          (** Set limits to all devices in the group **)
          IF GVL.UseTempGroupInputs AND (baseIdx - 10) + 6 < SIZEOF(GVL.TempGroupInput) / SIZEOF(GVL.TempGroupInput[0]) THEN
            THIS^.VoutSetMin[devIdx] := GVL.TempGroupInput[(baseIdx - 10) + 3];
            THIS^.VoutSetMax[devIdx] := GVL.TempGroupInput[(baseIdx - 10) + 4];
            THIS^.IoutSetMin[devIdx] := GVL.TempGroupInput[(baseIdx - 10) + 5];
            THIS^.IoutSetMax[devIdx] := MIN(GVL.TempGroupInput[(baseIdx - 10) + 6], GVL.GroupCapacity[groupIdx]);
          ELSE
            THIS^.VoutSetMin[devIdx] := GVL.NumericInput[baseIdx + 3]; (** GroupVoutSetMin **)
            THIS^.VoutSetMax[devIdx] := GVL.NumericInput[baseIdx + 4]; (** GroupVoutSetMax **)
            THIS^.IoutSetMin[devIdx] := GVL.NumericInput[baseIdx + 5]; (** GroupIoutSetMin **)
            THIS^.IoutSetMax[devIdx] := MIN(GVL.NumericInput[baseIdx + 6], GVL.GroupCapacity[groupIdx]); (** GroupIoutSetMax, constrained by min(GroupIoutSetMax, GroupCapacity) **)
          END_IF;
          
          (** Queue commands for group flags if changed **)
          IF GVL.Direction[devIdx] <> THIS^.LastDirection[devIdx] THEN
            IF THIS^.ApplyCommands(devIdx, GVL_Constant.CMD_DIRECTION_CTRL, BOOL_TO_UINT(GVL.Direction[devIdx])) THEN (** CMD_DIRECTION_CTRL **)
              THIS^.LastDirection[devIdx] := GVL.Direction[devIdx];
            END_IF;
          END_IF;
          
          IF GVL.OperationOn[devIdx] <> THIS^.LastOperationOn[devIdx] THEN
            IF THIS^.ApplyCommands(devIdx, GVL_Constant.CMD_OPERATION, BOOL_TO_UINT(GVL.OperationOn[devIdx])) THEN (** CMD_OPERATION **)
              THIS^.LastOperationOn[devIdx] := GVL.OperationOn[devIdx];
            END_IF;
          END_IF;
        END_IF;
      END_FOR;
    END_IF;
  END_IF;
END_FOR;

(** Process device inputs and queue control commands **)
FOR devIdx := 0 TO 19 DO
  baseIdx := 38 + (devIdx * 7); (** Device inputs start at 38 **)
  
  (** Read device setpoints and flags **)
  IF baseIdx + 6 < SIZEOF(GVL.NumericInput) / SIZEOF(GVL.NumericInput[0]) THEN
    (** Set setpoints for non-master devices or in maintenance mode **)
    IF GVL.UseTempBus1Direct AND devIdx <= 3 THEN
      GVL.VoutSetpoint[devIdx] := UINT_TO_REAL(GVL.TempBus1VoutSetpoint[devIdx]); (** Temp Bus1 VoutSetpoint **)
      GVL.IoutSetpoint[devIdx] := UINT_TO_REAL(GVL.TempBus1IoutSetpoint[devIdx]); (** Temp Bus1 IoutSetpoint **)
    ELSIF maintenanceMode OR devIdx < 4 OR GVL.GroupMembership[devIdx] = -1 OR NOT (GVL.GroupMaster[GVL.GroupMembership[devIdx]] = devIdx) THEN
      GVL.VoutSetpoint[devIdx] := UINT_TO_REAL(GVL.NumericInput[baseIdx]); (** VoutSetpoint **)
      GVL.IoutSetpoint[devIdx] := UINT_TO_REAL(GVL.NumericInput[baseIdx + 1]); (** IoutSetpoint **)
    END_IF;
    IF GVL.UseTempBus1Direct AND devIdx <= 3 THEN
      flags := GVL.TempBus1Flags[devIdx]; (** Temp Bus1 device flags **)
    ELSE
      flags := GVL.NumericInput[baseIdx + 2]; (** Device flags **)
    END_IF;
    
    (** Set device flags in maintenance mode or for devices 0-3 or non-master devices **)
    IF GVL.UseTempBus1Direct AND devIdx <= 3 THEN
      GVL.Voltage[devIdx] := (flags AND 16#0008) <> 0; (** Bit 3: DeviceMode Voltage **)
      GVL.Current[devIdx] := (flags AND 16#0004) <> 0; (** Bit 2: DeviceMode Current **)
      GVL.Standby[devIdx] := NOT (GVL.Voltage[devIdx] OR GVL.Current[devIdx]); (** Standby when neither Voltage nor Current **)
      GVL.Direction[devIdx] := (flags AND 16#0001) <> 0; (** Bit 0: Direction **)
      GVL.OperationOn[devIdx] := (flags AND 16#0002) <> 0; (** Bit 1: OperationOn **)
      GVL.OutputOn[devIdx] := (flags AND 16#0010) <> 0; (** Bit 4: OutputOn **)
    ELSIF maintenanceMode OR devIdx < 4 OR GVL.GroupMembership[devIdx] = -1 OR NOT (GVL.GroupMaster[GVL.GroupMembership[devIdx]] = devIdx) THEN
      GVL.Voltage[devIdx] := (flags AND 16#0008) <> 0; (** Bit 3: DeviceMode Voltage **)
      GVL.Current[devIdx] := (flags AND 16#0004) <> 0; (** Bit 2: DeviceMode Current **)
      GVL.Standby[devIdx] := NOT (GVL.Voltage[devIdx] OR GVL.Current[devIdx]); (** Standby when neither Voltage nor Current **)
      GVL.Direction[devIdx] := (flags AND 16#0001) <> 0; (** Bit 0: Direction **)
      GVL.OperationOn[devIdx] := (flags AND 16#0002) <> 0; (** Bit 1: OperationOn **)
      GVL.OutputOn[devIdx] := (flags AND 16#0010) <> 0; (** Bit 4: OutputOn **)
    END_IF;
    GVL.OrangeStop[devIdx] := (flags AND 16#0020) <> 0; (** Bit 5: OrangeStop **)
    GVL.RedStop[devIdx] := (flags AND 16#0040) <> 0; (** Bit 6: RedStop **)
    GVL.EStop[devIdx] := (flags AND 16#0080) <> 0; (** Bit 7: EStop **)
  END_IF;

  (** Queue direction command if requested direction differs from device feedback **)
  IF (GVL.UseTempBus1Direct AND devIdx <= 3 AND GVL.Direction[devIdx] <> THIS^.LastDirection[devIdx]) OR
     (NOT (GVL.UseTempBus1Direct AND devIdx <= 3) AND (GVL.Direction[devIdx] <> ((GVL.DeviceSystemFlags[devIdx] AND 16#0008) <> 0) OR 
     GVL.Direction[devIdx] <> THIS^.LastDirection[devIdx])) THEN
    IF THIS^.ApplyCommands(devIdx, GVL_Constant.CMD_DIRECTION_CTRL, BOOL_TO_UINT(GVL.Direction[devIdx])) THEN (** CMD_DIRECTION_CTRL **)
      THIS^.LastDirection[devIdx] := GVL.Direction[devIdx];
    END_IF;
  END_IF;

  (** Queue operation command **)
  IF GVL.OperationOn[devIdx] <> THIS^.LastOperationOn[devIdx] THEN
    IF THIS^.ApplyCommands(devIdx, GVL_Constant.CMD_OPERATION, BOOL_TO_UINT(GVL.OperationOn[devIdx])) THEN (** CMD_OPERATION **)
      THIS^.LastOperationOn[devIdx] := GVL.OperationOn[devIdx];
    END_IF;
  END_IF;

  (** Queue setpoint commands based on DeviceMode and Direction **)
  IF GVL.Standby[devIdx] THEN
    (** Standby mode **)
    IF THIS^.LastVoutSetpoint[devIdx] <> 0 THEN
      IF GVL.Direction[devIdx] THEN
        IF THIS^.ApplyCommands(devIdx, GVL_Constant.CMD_REVERSE_VOUT_SET, 0) THEN (** CMD_REVERSE_VOUT_SET, 0 **)
          GVL.VoutSetRev[devIdx] := 0.0; (** Clear reverse Vout setpoint **)
          THIS^.LastVoutSetpoint[devIdx] := 0;
        END_IF;
      ELSE
        IF THIS^.ApplyCommands(devIdx, GVL_Constant.CMD_VOUT_SET, 0) THEN (** CMD_VOUT_SET, 0 **)
          GVL.VoutSetpoint[devIdx] := 0.0; (** Clear forward Vout setpoint **)
          THIS^.LastVoutSetpoint[devIdx] := 0;
        END_IF;
      END_IF;
    END_IF;
    IF THIS^.LastIoutSetpoint[devIdx] <> 0 THEN
      IF GVL.Direction[devIdx] THEN
        IF THIS^.ApplyCommands(devIdx, GVL_Constant.CMD_REVERSE_IOUT_SET, 0) THEN (** CMD_REVERSE_IOUT_SET, 0 **)
          GVL.IoutSetRev[devIdx] := 0.0; (** Clear reverse Iout setpoint **)
          THIS^.LastIoutSetpoint[devIdx] := 0;
        END_IF;
      ELSE
        IF THIS^.ApplyCommands(devIdx, GVL_Constant.CMD_IOUT_SET, 0) THEN (** CMD_IOUT_SET, 0 **)
          GVL.IoutSetpoint[devIdx] := 0.0; (** Clear forward Iout setpoint **)
          THIS^.LastIoutSetpoint[devIdx] := 0;
        END_IF;
      END_IF;
    END_IF;
  ELSIF GVL.Current[devIdx] THEN
    (** Current mode **)
    setpointIout := MIN(MAX(GVL.IoutSetpoint[devIdx]/100, UINT_TO_REAL(THIS^.IoutSetMin[devIdx])), UINT_TO_REAL(THIS^.IoutSetMax[devIdx])); (** Clamp in native units **)
    IF devIdx <= 3 THEN
      clampedIout := REAL_TO_UINT(setpointIout * 10.0);   (** DPU F=0.1 **)
    ELSE
      factorNibble := SHR((GVL.VoutScale[devIdx] AND 16#00F0), 4);
      CASE factorNibble OF
        16#4: clampedIout := REAL_TO_UINT(setpointIout * 1000.0);
        16#5: clampedIout := REAL_TO_UINT(setpointIout * 100.0);
        16#6: clampedIout := REAL_TO_UINT(setpointIout * 10.0);
        16#7: clampedIout := REAL_TO_UINT(setpointIout);
        16#8: clampedIout := REAL_TO_UINT(setpointIout * 0.1);
        16#9: clampedIout := REAL_TO_UINT(setpointIout * 0.01);
        ELSE clampedIout := REAL_TO_UINT(setpointIout * 100.0);
      END_CASE;
    END_IF;
    IF clampedIout <> THIS^.LastIoutSetpoint[devIdx] THEN
      IF GVL.Direction[devIdx] THEN
        IF THIS^.ApplyCommands(devIdx, GVL_Constant.CMD_REVERSE_IOUT_SET, clampedIout) THEN (** CMD_REVERSE_IOUT_SET **)
          THIS^.LastIoutSetpoint[devIdx] := clampedIout;
        END_IF;
      ELSE
        IF THIS^.ApplyCommands(devIdx, GVL_Constant.CMD_IOUT_SET, clampedIout) THEN (** CMD_IOUT_SET **)
          THIS^.LastIoutSetpoint[devIdx] := clampedIout;
        END_IF;
      END_IF;
    END_IF;
  ELSIF GVL.Voltage[devIdx] THEN
    (** Voltage mode **)
    setpointVout := MIN(MAX(GVL.VoutSetpoint[devIdx]/100, UINT_TO_REAL(THIS^.VoutSetMin[devIdx])), UINT_TO_REAL(THIS^.VoutSetMax[devIdx])); (** Clamp in native units **)
    IF devIdx <= 3 THEN
      clampedVout := REAL_TO_UINT(setpointVout * 10.0);   (** DPU F=0.1 **)
    ELSE
      factorNibble := GVL.VoutScale[devIdx] AND 16#000F;
      CASE factorNibble OF
        16#4: clampedVout := REAL_TO_UINT(setpointVout * 1000.0);
        16#5: clampedVout := REAL_TO_UINT(setpointVout * 100.0);
        16#6: clampedVout := REAL_TO_UINT(setpointVout * 10.0);
        16#7: clampedVout := REAL_TO_UINT(setpointVout);
        16#8: clampedVout := REAL_TO_UINT(setpointVout * 0.1);
        16#9: clampedVout := REAL_TO_UINT(setpointVout * 0.01);
        ELSE clampedVout := REAL_TO_UINT(setpointVout * 100.0);
      END_CASE;
    END_IF;
    IF clampedVout <> THIS^.LastVoutSetpoint[devIdx] THEN
      IF GVL.Direction[devIdx] THEN
        IF THIS^.ApplyCommands(devIdx, GVL_Constant.CMD_REVERSE_VOUT_SET, clampedVout) THEN (** CMD_REVERSE_VOUT_SET **)
          THIS^.LastVoutSetpoint[devIdx] := clampedVout;
        END_IF;
      ELSE
        IF THIS^.ApplyCommands(devIdx, GVL_Constant.CMD_VOUT_SET, clampedVout) THEN (** CMD_VOUT_SET **)
          THIS^.LastVoutSetpoint[devIdx] := clampedVout;
        END_IF;
      END_IF;
    END_IF;
  END_IF;
END_FOR;
END_METHOD

METHOD ReadLimits
VAR
  devIdx : INT;                            (* Device index *)
  baseIdx : INT;                           (* Base index for device inputs *)
  inputIdx : INT;                          (* Base index for group inputs *)
  groupIdx : INT;                          (* Group index *)
  masterIdx : INT;                         (* Master device index *)
  maintenanceMode : BOOL;                  (* Maintenance mode status *)
  tempBase : INT;                          (* Temp: offset into TempGroupInput array *)
END_VAR

(* Comment Section: GVL.NumericInput Mapping for ReadLimits *)
(* This method reads individual setpoints/limits for all devices and applies *)
(* group-level setpoints/limits to the master device in normal mode. Group limits *)
(* (e.g., GroupIoutSetMax) are constrained by GVL.GroupCapacity, set by GroupManager *)
(* based on healthy units. GVL.GroupMaster serves as the group device index, *)
(* enabling groups when valid (4-19). *)

(* GVL.NumericInput Mapping *)
(* 0-4: System-Level Inputs *)
(*   0: GVL.SystemAlarms *)
(*   1: System Flags (maintenanceMode read here) *)
(*   2: Morphee Signal *)
(*   3-4: Reserved *)
(* 5-9: Unallocated *)
(* 10-37: Group Inputs (4 groups x 7 inputs) *)
(*   - For groupIdx = 0 TO 3, baseIdx = 10 + (groupIdx * 7): *)
(*     baseIdx: GroupVoutSetpoint *)
(*     baseIdx + 1: GroupIoutSetpoint *)
(*     baseIdx + 2: Group Flags *)
(*     baseIdx + 3: GroupVoutSetMin *)
(*     baseIdx + 4: GroupVoutSetMax *)
(*     baseIdx + 5: GroupIoutSetMin *)
(*     baseIdx + 6: GroupIoutSetMax *)
(*   - Applied to master device here if valid *)
(* 38-177: Device Inputs (20 devices x 7 inputs) *)
(*   - For devIdx = 0 TO 19, baseIdx = 38 + (devIdx * 7): *)
(*     baseIdx: VoutSetpoint *)
(*     baseIdx + 1: IoutSetpoint *)
(*     baseIdx + 2: Flags *)
(*     baseIdx + 3: VoutSetMin *)
(*     baseIdx + 4: VoutSetMax *)
(*     baseIdx + 5: IoutSetMin *)
(*     baseIdx + 6: IoutSetMax *)
(* 178+: Unallocated *)

(* Read maintenance mode *)
maintenanceMode := (GVL.NumericInput[1] AND 16#0001) <> 0; (* Index 1, bit 0 *)

(* Set individual device setpoints and limits *)
FOR devIdx := 0 TO 19 DO
  baseIdx := 38 + (devIdx * 7);
  IF baseIdx + 6 < SIZEOF(GVL.NumericInput) / SIZEOF(GVL.NumericInput[0]) THEN
    IF GVL.UseTempBus1Direct AND devIdx <= 3 THEN
      VoutSetpoint[devIdx] := GVL.TempBus1VoutSetpoint[devIdx];
      IoutSetpoint[devIdx] := GVL.TempBus1IoutSetpoint[devIdx];
      VoutSetMin[devIdx] := GVL.TempBus1VoutSetMin[devIdx] / 100;
      VoutSetMax[devIdx] := GVL.TempBus1VoutSetMax[devIdx] / 100;
      IoutSetMin[devIdx] := GVL.TempBus1IoutSetMin[devIdx] / 100;
      IoutSetMax[devIdx] := GVL.TempBus1IoutSetMax[devIdx] / 100;
    ELSE
      VoutSetpoint[devIdx] := GVL.NumericInput[baseIdx];
      IoutSetpoint[devIdx] := GVL.NumericInput[baseIdx + 1];
      VoutSetMin[devIdx] := GVL.NumericInput[baseIdx + 3];
      VoutSetMax[devIdx] := GVL.NumericInput[baseIdx + 4];
      IoutSetMin[devIdx] := GVL.NumericInput[baseIdx + 5];
      IoutSetMax[devIdx] := GVL.NumericInput[baseIdx + 6];
    END_IF;
  END_IF;

  (* Apply group-level setpoints and limits to master in normal mode *)
  IF NOT maintenanceMode AND devIdx >= 4 THEN
    FOR groupIdx := 0 TO 3 DO
      masterIdx := GVL.GroupMaster[groupIdx];
      IF masterIdx >= 4 AND masterIdx <= 19 AND NOT GVL.SafetyShutdown[masterIdx] THEN
        CASE groupIdx OF
          0: inputIdx := 10; (* LVLA1 *)
          1: inputIdx := 17; (* LVLA2 *)
          2: inputIdx := 24; (* LVLA3 *)
          3: inputIdx := 31; (* LVLA4 *)
        END_CASE;
        IF devIdx = masterIdx THEN
          IF inputIdx + 6 < SIZEOF(GVL.NumericInput) / SIZEOF(GVL.NumericInput[0]) THEN
            IF GVL.UseTempGroupInputs THEN
              tempBase := inputIdx - 10; (* Map group base (10..) to TempGroupInput (0..) *)
              IF tempBase >= 0 AND tempBase + 6 < SIZEOF(GVL.TempGroupInput) / SIZEOF(GVL.TempGroupInput[0]) THEN
                VoutSetpoint[masterIdx] := GVL.TempGroupInput[tempBase];
                IoutSetpoint[masterIdx] := GVL.TempGroupInput[tempBase + 1];
                VoutSetMin[masterIdx] := GVL.TempGroupInput[tempBase + 3];
                VoutSetMax[masterIdx] := GVL.TempGroupInput[tempBase + 4];
                IoutSetMin[masterIdx] := GVL.TempGroupInput[tempBase + 5];
                IoutSetMax[masterIdx] := MIN(GVL.TempGroupInput[tempBase + 6], GVL.GroupCapacity[groupIdx]); (* Constrain by capacity *)
              END_IF;
            ELSE
              VoutSetpoint[masterIdx] := GVL.NumericInput[inputIdx];
              IoutSetpoint[masterIdx] := GVL.NumericInput[inputIdx + 1];
              VoutSetMin[masterIdx] := GVL.NumericInput[inputIdx + 3];
              VoutSetMax[masterIdx] := GVL.NumericInput[inputIdx + 4];
              IoutSetMin[masterIdx] := GVL.NumericInput[inputIdx + 5];
              IoutSetMax[masterIdx] := MIN(GVL.NumericInput[inputIdx + 6], GVL.GroupCapacity[groupIdx]); (* Constrain by capacity *)
            END_IF;
          END_IF;
        END_IF;
      END_IF;
    END_FOR;
  END_IF;
END_FOR;
END_METHOD

METHOD UpdateOutputs
VAR
  devIdx : INT;                            (* Device index *)
  baseIdx : INT;                           (* Base index for output array *)
  systemAlarms : DWORD;                    (* System alarms for output *)
  maintenanceMode : BOOL;                  (* Maintenance mode status *)
  cmdId : BYTE;                            (* Command ID for init data *)
  cmdOffset : INT;                         (* Command offset for init frame *)
  i : INT;                                 (* Loop variable for commands *)
  j : INT;                                 (* Loop variable for data pairs *)
  idx : INT;                               (* Output array index *)
  watchDog : BOOL;                         (* Watchdog toggle for output *)
  updatingInMorpheeTableInprogress : Bool := FALSE;
  groupIdx : INT;                          (* Group index *)
  masterIdx : INT;                         (* Master device index *)
  groupBase : INT;                         (* Base index for group devices *)
  opCount : UINT;                          (* Count of devices with OperationOn *)
  outCount : UINT;                         (* Count of devices with OutputOn *)
  initTimeoutCounter : UINT;               (* Counter for forced init exit *)
  commandCount : UINT;                     (* Commands per cycle *)
  commandArray : ARRAY[0..8] OF BYTE := [16#80, 16#81, 16#82, 16#83, 16#84, 16#85, 16#86, 16#87, 16#88];
  commandIndex : INT;
  upperBound : INT;                        (* Upper bound for FOR loop *)
	scaledVin: INT; (** Scaled input voltage **)
	scaledVout: UINT; (** Scaled output voltage **)
	scaledIout: UINT; (** Scaled current **)
	scaledTemp: UINT; (** Scaled temperature **)
	scaledFanSpeed1: INT; (** Scaled fan speed 1 **)
	scaledFanSpeed2: INT; (** Scaled fan speed 2 **)
	scaledIin: INT; (** Scaled input current **)
	tempScale: UINT; (** Temporary variable for scaling factor extraction **)
	scaleValue: UINT; (** Extracted 4-bit scaling value **)
 
END_VAR
(* One-time reset of GVL variables *)
IF GVL.FirstRun THEN
    FOR devIdx := 0 TO 19 DO
        GVL.Voltage[devIdx] := FALSE;
        GVL.Current[devIdx] := FALSE;
        GVL.Standby[devIdx] := FALSE;
        GVL.OperationOn[devIdx] := FALSE;
        GVL.Direction[devIdx] := FALSE;
        GVL.OutputOn[devIdx] := FALSE;
        GVL.OrangeStop[devIdx] := FALSE;
        GVL.RedStop[devIdx] := FALSE;
        GVL.EStop[devIdx] := FALSE;
        GVL.Vin[devIdx] := 0;
        GVL.Vout[devIdx] := 0;
        GVL.Iout[devIdx] := 0;
        GVL.Temperature[devIdx] := 0;
        GVL.FanSpeed1[devIdx] := 0;
        GVL.FanSpeed2[devIdx] := 0;
        GVL.Iin[devIdx] := 0;
        GVL.FaultStatus[devIdx] := 0;
        GVL.TemperatureFaultHigh[devIdx] := FALSE;
        CanCtrlConfigured[devIdx] := FALSE;
    END_FOR;
    GVL.FirstRun := FALSE;
END_IF;

watchDog := NOT watchDog;


// Detect Morphee initialization request (GVL.NumericInput[2] changes)
IF GVL.NumericInput[2] <> LastMorpheeSignal AND NOT updatingInMorpheeTableInprogress THEN
    LastMorpheeSignal := DWORD_TO_UINT(GVL.NumericInput[2]);
    CASE GVL.NumericInput[2] OF
        1..6: // Morphee requests initialization cycles 1 to 6
            IsInitPhase := TRUE;
            InitCycle := DWORD_TO_UINT(GVL.NumericInput[2]);
            initTimeoutCounter := 0;
            InitTimeout(IN := FALSE);
        100: // Morphee signals completion
            IsInitPhase := FALSE;
            InitCycle := 0;
            initTimeoutCounter := 0;
            InitTimeout(IN := FALSE);
    END_CASE;
END_IF;

(* In temporary setpoint test mode, keep normal output update path active. *)
IF GVL.UseTempGroupInputs THEN
  IsInitPhase := FALSE;
  InitCycle := 0;
END_IF;

// Initialization phase logic
IF IsInitPhase THEN
    initTimeoutCounter := initTimeoutCounter + 1;
    // Remove strict timeout to ensure all cycles complete
    // IF initTimeoutCounter > 1000 THEN
    //     IsInitPhase := FALSE;
    //     InitCycle := 0;
    //     initTimeoutCounter := 0;
    //     InitTimeout(IN := FALSE);
    // END_IF;

    InitTimeout(IN := TRUE, PT := T#100MS);

    IF InitCycle > 0 AND IsInitPhase THEN
        updatingInMorpheeTableInprogress := TRUE;
        FOR devIdx := 0 TO 19 DO
            idx := devIdx * 6; // Base index for the device
            IF idx + 5 < 120 THEN // Ensure within array bounds
                CASE InitCycle OF
                    1: // 0x80 and 0x81 (bytes 0-11)
                        cmdId := 16#80;
                        baseIdx := 0;
                        IF baseIdx + 1 < 54 THEN
                            GVL.NumericOutput[idx] := SHL(TO_DWORD(cmdId), 24) OR SHL(TO_DWORD(devIdx), 16) OR SHL(TO_DWORD(GVL.MfrSerialPersistent[devIdx][baseIdx]), 8) OR TO_DWORD(GVL.MfrSerialPersistent[devIdx][baseIdx + 1]);
                            GVL.NumericOutput[idx + 1] := SHL(TO_DWORD(cmdId), 24) OR SHL(TO_DWORD(devIdx), 16) OR SHL(TO_DWORD(GVL.MfrSerialPersistent[devIdx][baseIdx + 2]), 8) OR TO_DWORD(GVL.MfrSerialPersistent[devIdx][baseIdx + 3]);
                            GVL.NumericOutput[idx + 2] := SHL(TO_DWORD(cmdId), 24) OR SHL(TO_DWORD(devIdx), 16) OR SHL(TO_DWORD(GVL.MfrSerialPersistent[devIdx][baseIdx + 4]), 8) OR TO_DWORD(GVL.MfrSerialPersistent[devIdx][baseIdx + 5]);
                        END_IF;
                        cmdId := 16#81;
                        baseIdx := 6;
                        IF baseIdx + 1 < 54 THEN
                            GVL.NumericOutput[idx + 3] := SHL(TO_DWORD(cmdId), 24) OR SHL(TO_DWORD(devIdx), 16) OR SHL(TO_DWORD(GVL.MfrSerialPersistent[devIdx][baseIdx]), 8) OR TO_DWORD(GVL.MfrSerialPersistent[devIdx][baseIdx + 1]);
                            GVL.NumericOutput[idx + 4] := SHL(TO_DWORD(cmdId), 24) OR SHL(TO_DWORD(devIdx), 16) OR SHL(TO_DWORD(GVL.MfrSerialPersistent[devIdx][baseIdx + 2]), 8) OR TO_DWORD(GVL.MfrSerialPersistent[devIdx][baseIdx + 3]);
                            GVL.NumericOutput[idx + 5] := SHL(TO_DWORD(cmdId), 24) OR SHL(TO_DWORD(devIdx), 16) OR SHL(TO_DWORD(GVL.MfrSerialPersistent[devIdx][baseIdx + 4]), 8) OR TO_DWORD(GVL.MfrSerialPersistent[devIdx][baseIdx + 5]);
                        END_IF;
                    2: // 0x82 and 0x83 (bytes 12-23)
                        cmdId := 16#82;
                        baseIdx := 12;
                        IF baseIdx + 1 < 54 THEN
                            GVL.NumericOutput[idx] := SHL(TO_DWORD(cmdId), 24) OR SHL(TO_DWORD(devIdx), 16) OR SHL(TO_DWORD(GVL.MfrSerialPersistent[devIdx][baseIdx]), 8) OR TO_DWORD(GVL.MfrSerialPersistent[devIdx][baseIdx + 1]);
                            GVL.NumericOutput[idx + 1] := SHL(TO_DWORD(cmdId), 24) OR SHL(TO_DWORD(devIdx), 16) OR SHL(TO_DWORD(GVL.MfrSerialPersistent[devIdx][baseIdx + 2]), 8) OR TO_DWORD(GVL.MfrSerialPersistent[devIdx][baseIdx + 3]);
                            GVL.NumericOutput[idx + 2] := SHL(TO_DWORD(cmdId), 24) OR SHL(TO_DWORD(devIdx), 16) OR SHL(TO_DWORD(GVL.MfrSerialPersistent[devIdx][baseIdx + 4]), 8) OR TO_DWORD(GVL.MfrSerialPersistent[devIdx][baseIdx + 5]);
                        END_IF;
                        cmdId := 16#83;
                        baseIdx := 18;
                        IF baseIdx + 1 < 54 THEN
                            GVL.NumericOutput[idx + 3] := SHL(TO_DWORD(cmdId), 24) OR SHL(TO_DWORD(devIdx), 16) OR SHL(TO_DWORD(GVL.MfrSerialPersistent[devIdx][baseIdx]), 8) OR TO_DWORD(GVL.MfrSerialPersistent[devIdx][baseIdx + 1]);
                            GVL.NumericOutput[idx + 4] := SHL(TO_DWORD(cmdId), 24) OR SHL(TO_DWORD(devIdx), 16) OR SHL(TO_DWORD(GVL.MfrSerialPersistent[devIdx][baseIdx + 2]), 8) OR TO_DWORD(GVL.MfrSerialPersistent[devIdx][baseIdx + 3]);
                            GVL.NumericOutput[idx + 5] := SHL(TO_DWORD(cmdId), 24) OR SHL(TO_DWORD(devIdx), 16) OR SHL(TO_DWORD(GVL.MfrSerialPersistent[devIdx][baseIdx + 4]), 8) OR TO_DWORD(GVL.MfrSerialPersistent[devIdx][baseIdx + 5]);
                        END_IF;
                    3: // 0x84 (bytes 24-29)
                        cmdId := 16#84;
                        baseIdx := 24;
                        IF baseIdx + 1 < 54 THEN
                            GVL.NumericOutput[idx] := SHL(TO_DWORD(cmdId), 24) OR SHL(TO_DWORD(devIdx), 16) OR SHL(TO_DWORD(GVL.MfrSerialPersistent[devIdx][baseIdx]), 8) OR TO_DWORD(GVL.MfrSerialPersistent[devIdx][baseIdx + 1]);
                            GVL.NumericOutput[idx + 1] := SHL(TO_DWORD(cmdId), 24) OR SHL(TO_DWORD(devIdx), 16) OR SHL(TO_DWORD(GVL.MfrSerialPersistent[devIdx][baseIdx + 2]), 8) OR TO_DWORD(GVL.MfrSerialPersistent[devIdx][baseIdx + 3]);
                            GVL.NumericOutput[idx + 2] := SHL(TO_DWORD(cmdId), 24) OR SHL(TO_DWORD(devIdx), 16) OR SHL(TO_DWORD(GVL.MfrSerialPersistent[devIdx][baseIdx + 4]), 8) OR TO_DWORD(GVL.MfrSerialPersistent[devIdx][baseIdx + 5]);
                        END_IF;
                    4: // 0x85 (bytes 30-35)
                        cmdId := 16#85;
                        baseIdx := 30;
                        IF baseIdx + 1 < 54 THEN
                            GVL.NumericOutput[idx] := SHL(TO_DWORD(cmdId), 24) OR SHL(TO_DWORD(devIdx), 16) OR SHL(TO_DWORD(GVL.MfrSerialPersistent[devIdx][baseIdx]), 8) OR TO_DWORD(GVL.MfrSerialPersistent[devIdx][baseIdx + 1]);
                            GVL.NumericOutput[idx + 1] := SHL(TO_DWORD(cmdId), 24) OR SHL(TO_DWORD(devIdx), 16) OR SHL(TO_DWORD(GVL.MfrSerialPersistent[devIdx][baseIdx + 2]), 8) OR TO_DWORD(GVL.MfrSerialPersistent[devIdx][baseIdx + 3]);
                            GVL.NumericOutput[idx + 2] := SHL(TO_DWORD(cmdId), 24) OR SHL(TO_DWORD(devIdx), 16) OR SHL(TO_DWORD(GVL.MfrSerialPersistent[devIdx][baseIdx + 4]), 8) OR TO_DWORD(GVL.MfrSerialPersistent[devIdx][baseIdx + 5]);
                        END_IF;
                    5: // 0x86 (bytes 36-41)
                        cmdId := 16#86;
                        baseIdx := 36;
                        IF baseIdx + 1 < 54 THEN
                            GVL.NumericOutput[idx] := SHL(TO_DWORD(cmdId), 24) OR SHL(TO_DWORD(devIdx), 16) OR SHL(TO_DWORD(GVL.MfrSerialPersistent[devIdx][baseIdx]), 8) OR TO_DWORD(GVL.MfrSerialPersistent[devIdx][baseIdx + 1]);
                            GVL.NumericOutput[idx + 1] := SHL(TO_DWORD(cmdId), 24) OR SHL(TO_DWORD(devIdx), 16) OR SHL(TO_DWORD(GVL.MfrSerialPersistent[devIdx][baseIdx + 2]), 8) OR TO_DWORD(GVL.MfrSerialPersistent[devIdx][baseIdx + 3]);
                            GVL.NumericOutput[idx + 2] := SHL(TO_DWORD(cmdId), 24) OR SHL(TO_DWORD(devIdx), 16) OR SHL(TO_DWORD(GVL.MfrSerialPersistent[devIdx][baseIdx + 4]), 8) OR TO_DWORD(GVL.MfrSerialPersistent[devIdx][baseIdx + 5]);
                        END_IF;
                    6: // 0x87 and 0x88 (bytes 42-53)
                        cmdId := 16#87;
                        baseIdx := 42;
                        IF baseIdx + 1 < 54 THEN
                            GVL.NumericOutput[idx] := SHL(TO_DWORD(cmdId), 24) OR SHL(TO_DWORD(devIdx), 16) OR SHL(TO_DWORD(GVL.MfrSerialPersistent[devIdx][baseIdx]), 8) OR TO_DWORD(GVL.MfrSerialPersistent[devIdx][baseIdx + 1]);
                            GVL.NumericOutput[idx + 1] := SHL(TO_DWORD(cmdId), 24) OR SHL(TO_DWORD(devIdx), 16) OR SHL(TO_DWORD(GVL.MfrSerialPersistent[devIdx][baseIdx + 2]), 8) OR TO_DWORD(GVL.MfrSerialPersistent[devIdx][baseIdx + 3]);
                            GVL.NumericOutput[idx + 2] := SHL(TO_DWORD(cmdId), 24) OR SHL(TO_DWORD(devIdx), 16) OR SHL(TO_DWORD(GVL.MfrSerialPersistent[devIdx][baseIdx + 4]), 8) OR TO_DWORD(GVL.MfrSerialPersistent[devIdx][baseIdx + 5]);
                        END_IF;
                        cmdId := 16#88;
                        baseIdx := 48;
                        IF baseIdx + 1 < 54 THEN
                            GVL.NumericOutput[idx + 3] := SHL(TO_DWORD(cmdId), 24) OR SHL(TO_DWORD(devIdx), 16) OR SHL(TO_DWORD(GVL.MfrSerialPersistent[devIdx][baseIdx]), 8) OR TO_DWORD(GVL.MfrSerialPersistent[devIdx][baseIdx + 1]);
                            GVL.NumericOutput[idx + 4] := SHL(TO_DWORD(cmdId), 24) OR SHL(TO_DWORD(devIdx), 16) OR SHL(TO_DWORD(GVL.MfrSerialPersistent[devIdx][baseIdx + 2]), 8) OR TO_DWORD(GVL.MfrSerialPersistent[devIdx][baseIdx + 3]);
                            GVL.NumericOutput[idx + 5] := SHL(TO_DWORD(cmdId), 24) OR SHL(TO_DWORD(devIdx), 16) OR SHL(TO_DWORD(GVL.MfrSerialPersistent[devIdx][baseIdx + 4]), 8) OR TO_DWORD(GVL.MfrSerialPersistent[devIdx][baseIdx + 5]);
                        END_IF;
                END_CASE;
            END_IF;
        END_FOR;
        updatingInMorpheeTableInprogress := FALSE;
    END_IF;
ELSE
    updatingInMorpheeTableInprogress := FALSE;
    InitTimeout(IN := FALSE);
    systemAlarms := UINT_TO_DWORD(GVL.SystemAlarms);
    maintenanceMode := (GVL.NumericInput[1] AND 16#0001) <> 0;

    FOR devIdx := 0 TO 19 DO
        baseIdx := devIdx * 5;
        // IF baseIdx < SIZEOF(GVL.NumericOutput) / SIZEOF(GVL.NumericOutput[0]) THEN
            (* Check for RedStop condition *)
            IF GVL.RedStop[devIdx] THEN
                GVL.Voltage[devIdx] := FALSE;
                GVL.Current[devIdx] := FALSE;
                GVL.Standby[devIdx] := TRUE;
                GVL.OperationOn[devIdx] := FALSE;
                GVL.Direction[devIdx] := FALSE;
                GVL.OutputOn[devIdx] := FALSE;
                GVL.OrangeStop[devIdx] := FALSE;
            END_IF;

            IF devIdx <= 3 THEN
              (* DPU fixed scaling from manual: VIN F=1, VOUT/IOUT/TEMP F=0.1, FAN F=1 *)
              scaledVin := GVL.Vin[devIdx];
              scaledVout := REAL_TO_UINT(UINT_TO_REAL(GVL.Vout[devIdx]) * 0.1);
            ELSE
              (* Scale GVL.Vin[devIdx] using VIN scaling factor, byte 1 bits 0-3 *)
              tempScale := GVL.VinScale[devIdx] AND 16#0F; (* Extract bits 0-3 *)
              IF tempScale = 16#4 THEN
                scaledVin := REAL_TO_UINT(UINT_TO_REAL(GVL.Vin[devIdx]) * 0.001);
              ELSIF tempScale = 16#5 THEN
                scaledVin := REAL_TO_UINT(UINT_TO_REAL(GVL.Vin[devIdx]) * 0.01);
              ELSIF tempScale = 16#6 THEN
                scaledVin := REAL_TO_UINT(UINT_TO_REAL(GVL.Vin[devIdx]) * 0.1);
              ELSIF tempScale = 16#7 THEN
                scaledVin := GVL.Vin[devIdx];
              ELSIF tempScale = 16#8 THEN
                scaledVin := REAL_TO_UINT(UINT_TO_REAL(GVL.Vin[devIdx]) * 10.0);
              ELSIF tempScale = 16#9 THEN
                scaledVin := REAL_TO_UINT(UINT_TO_REAL(GVL.Vin[devIdx]) * 100.0);
              ELSE
                scaledVin := REAL_TO_UINT(UINT_TO_REAL(GVL.Vin[devIdx]) * 0.1);
              END_IF;

              (* Scale GVL.Vout[devIdx] using VOUT scaling factor, byte 0 bits 0-3 *)
              tempScale := GVL.VoutScale[devIdx] AND 16#0F; (* Extract bits 0-3 *)
              IF tempScale = 16#4 THEN
                scaledVout := REAL_TO_UINT(UINT_TO_REAL(GVL.Vout[devIdx]) * 0.001);
              ELSIF tempScale = 16#5 THEN
                scaledVout := REAL_TO_UINT(UINT_TO_REAL(GVL.Vout[devIdx]) * 0.01);
              ELSIF tempScale = 16#6 THEN
                scaledVout := REAL_TO_UINT(UINT_TO_REAL(GVL.Vout[devIdx]) * 0.1);
              ELSIF tempScale = 16#7 THEN
                scaledVout := GVL.Vout[devIdx];
              ELSIF tempScale = 16#8 THEN
                scaledVout := REAL_TO_UINT(UINT_TO_REAL(GVL.Vout[devIdx]) * 10.0);
              ELSIF tempScale = 16#9 THEN
                scaledVout := REAL_TO_UINT(UINT_TO_REAL(GVL.Vout[devIdx]) * 100.0);
              ELSE
                scaledVout := REAL_TO_UINT(UINT_TO_REAL(GVL.Vout[devIdx]) * 0.1);
              END_IF;
            END_IF;

            IF GVL.Vin[devIdx] > 0 OR GVL.Vout[devIdx] > 0 THEN
              GVL.NumericOutput[baseIdx] := SHL(TO_DWORD(scaledVin), 16) OR TO_DWORD(scaledVout);
            ELSE
                GVL.NumericOutput[baseIdx] := 0;
            END_IF;

            IF devIdx <= 3 THEN
              scaledIout := REAL_TO_UINT(UINT_TO_REAL(GVL.Iout[devIdx]) * 0.1);
              scaledTemp := REAL_TO_UINT(UINT_TO_REAL(GVL.Temperature[devIdx]) * 0.1);
            ELSE
              (* Scale GVL.Iout[devIdx] using IOUT scaling factor, byte 0 bits 4-7 *)
              tempScale := GVL.VoutScale[devIdx] AND 16#F0; (* Mask bits 4-7 *)
              scaleValue := SHR(tempScale, 4); (* Shift right by 4 to get IOUT bits *)
              IF scaleValue = 16#4 THEN
                scaledIout := REAL_TO_UINT(UINT_TO_REAL(GVL.Iout[devIdx]) * 0.001);
              ELSIF scaleValue = 16#5 THEN
                scaledIout := REAL_TO_UINT(UINT_TO_REAL(GVL.Iout[devIdx]) * 0.01);
              ELSIF scaleValue = 16#6 THEN
                scaledIout := REAL_TO_UINT(UINT_TO_REAL(GVL.Iout[devIdx]) * 0.1);
              ELSIF scaleValue = 16#7 THEN
                scaledIout := GVL.Iout[devIdx];
              ELSIF scaleValue = 16#8 THEN
                scaledIout := REAL_TO_UINT(UINT_TO_REAL(GVL.Iout[devIdx]) * 10.0);
              ELSIF scaleValue = 16#9 THEN
                scaledIout := REAL_TO_UINT(UINT_TO_REAL(GVL.Iout[devIdx]) * 100.0);
              ELSE
                scaledIout := REAL_TO_UINT(UINT_TO_REAL(GVL.Iout[devIdx]) * 0.1);
              END_IF;

              (* Scale GVL.Temperature[devIdx] using TEMPERATURE_1 scaling factor, byte 2 bits 0-3 *)
              tempScale := GVL.TempScale[devIdx] AND 16#0F; (* Extract bits 0-3 *)
              IF tempScale = 16#4 THEN
                scaledTemp := REAL_TO_UINT(UINT_TO_REAL(GVL.Temperature[devIdx]) * 0.001);
              ELSIF tempScale = 16#5 THEN
                scaledTemp := REAL_TO_UINT(UINT_TO_REAL(GVL.Temperature[devIdx]) * 0.01);
              ELSIF tempScale = 16#6 THEN
                scaledTemp := REAL_TO_UINT(UINT_TO_REAL(GVL.Temperature[devIdx]) * 0.1);
              ELSIF tempScale = 16#7 THEN
                scaledTemp := GVL.Temperature[devIdx];
              ELSIF tempScale = 16#8 THEN
                scaledTemp := REAL_TO_UINT(UINT_TO_REAL(GVL.Temperature[devIdx]) * 10.0);
              ELSIF tempScale = 16#9 THEN
                scaledTemp := REAL_TO_UINT(UINT_TO_REAL(GVL.Temperature[devIdx]) * 100.0);
              ELSE
                scaledTemp := REAL_TO_UINT(UINT_TO_REAL(GVL.Temperature[devIdx]) * 0.1);
              END_IF;
            END_IF;

            (* Scale GVL.FanSpeed1[devIdx] and GVL.FanSpeed2[devIdx] using FAN_SPEED scaling factor, byte 1 bits 4-7 *)
            tempScale := GVL.VinScale[devIdx] AND 16#F0; (* Mask bits 4-7 *)
            scaleValue := SHR(tempScale, 4); (* Shift right by 4 to get FAN_SPEED bits *)
            IF scaleValue = 16#4 THEN
                scaledFanSpeed1 := REAL_TO_UINT(UINT_TO_REAL(GVL.FanSpeed1[devIdx]) * 0.001);
                scaledFanSpeed2 := REAL_TO_UINT(UINT_TO_REAL(GVL.FanSpeed2[devIdx]) * 0.001);
            ELSIF scaleValue = 16#5 THEN
                scaledFanSpeed1 := REAL_TO_UINT(UINT_TO_REAL(GVL.FanSpeed1[devIdx]) * 0.01);
                scaledFanSpeed2 := REAL_TO_UINT(UINT_TO_REAL(GVL.FanSpeed2[devIdx]) * 0.01);
            ELSIF scaleValue = 16#6 THEN
                scaledFanSpeed1 := REAL_TO_UINT(UINT_TO_REAL(GVL.FanSpeed1[devIdx]) * 0.1);
                scaledFanSpeed2 := REAL_TO_UINT(UINT_TO_REAL(GVL.FanSpeed2[devIdx]) * 0.1);
            ELSIF scaleValue = 16#7 THEN
                scaledFanSpeed1 := GVL.FanSpeed1[devIdx];
                scaledFanSpeed2 := GVL.FanSpeed2[devIdx];
            ELSIF scaleValue = 16#8 THEN
                scaledFanSpeed1 := REAL_TO_UINT(UINT_TO_REAL(GVL.FanSpeed1[devIdx]) * 10.0);
                scaledFanSpeed2 := REAL_TO_UINT(UINT_TO_REAL(GVL.FanSpeed2[devIdx]) * 10.0);
            ELSIF scaleValue = 16#9 THEN
                scaledFanSpeed1 := REAL_TO_UINT(UINT_TO_REAL(GVL.FanSpeed1[devIdx]) * 100.0);
                scaledFanSpeed2 := REAL_TO_UINT(UINT_TO_REAL(GVL.FanSpeed2[devIdx]) * 100.0);
            ELSE
                scaledFanSpeed1 := REAL_TO_UINT(UINT_TO_REAL(GVL.FanSpeed1[devIdx]) * 0.1);
                scaledFanSpeed2 := REAL_TO_UINT(UINT_TO_REAL(GVL.FanSpeed2[devIdx]) * 0.1);
            END_IF;

            (* Scale GVL.Iin[devIdx] using IIN scaling factor, byte 3 bits 0-3 *)
            tempScale := GVL.IinScale[devIdx] AND 16#0F; (* Extract bits 0-3 *)
            IF tempScale = 16#4 THEN
                scaledIin := REAL_TO_UINT(UINT_TO_REAL(GVL.Iin[devIdx]) * 0.001);
            ELSIF tempScale = 16#5 THEN
                scaledIin := REAL_TO_UINT(UINT_TO_REAL(GVL.Iin[devIdx]) * 0.01);
            ELSIF tempScale = 16#6 THEN
                scaledIin := REAL_TO_UINT(UINT_TO_REAL(GVL.Iin[devIdx]) * 0.1);
            ELSIF tempScale = 16#7 THEN
                scaledIin := GVL.Iin[devIdx];
            ELSIF tempScale = 16#8 THEN
                scaledIin := REAL_TO_UINT(UINT_TO_REAL(GVL.Iin[devIdx]) * 10.0);
            ELSIF tempScale = 16#9 THEN
                scaledIin := REAL_TO_UINT(UINT_TO_REAL(GVL.Iin[devIdx]) * 100.0);
            ELSE
                scaledIin := REAL_TO_UINT(UINT_TO_REAL(GVL.Iin[devIdx]) * 0.1);
            END_IF;

            GVL.NumericOutput[baseIdx + 1] := SHL(TO_DWORD(scaledIout), 16) OR TO_DWORD(scaledTemp);
            GVL.NumericOutput[baseIdx + 2] := SHL(TO_DWORD(scaledFanSpeed1), 16) OR TO_DWORD(scaledFanSpeed2);
            GVL.NumericOutput[baseIdx + 3] := SHL(TO_DWORD(GVL.FaultStatus[devIdx]), 16) OR 
                                              SHL(TO_DWORD(GVL.Direction[devIdx]), 0) OR 
                                              SHL(TO_DWORD(GVL.OperationOn[devIdx]), 1) OR 
                                              SHL(TO_DWORD(GVL.Current[devIdx]), 2) OR 
                                              SHL(TO_DWORD(GVL.Voltage[devIdx]), 3) OR 
                                              SHL(TO_DWORD(GVL.OutputOn[devIdx]), 4) OR 
                                              SHL(TO_DWORD(GVL.OrangeStop[devIdx]), 5) OR 
                                              SHL(TO_DWORD(GVL.RedStop[devIdx]), 6) OR 
                                              SHL(TO_DWORD(GVL.EStop[devIdx]), 7) OR 
                                              SHL(TO_DWORD(GVL.TemperatureFaultHigh[devIdx]), 8);
              GVL.NumericOutput[baseIdx + 4] := SHL(TO_DWORD(GVL.DeviceSystemFlags[devIdx]), 16);
        //END_IF;
    END_FOR;

    GVL.NumericOutput[100] := systemAlarms;
	 EL3174_Channel1_Alarm:=  EL3174_Channel1_value>(2.5*10)/32768;
 	 EL3174_Channel2_Alarm:=  EL3174_Channel2_value>(2.5*10)/32768;
 	 EL3174_Channel3_Alarm:=  EL3174_Channel3_value>(2.5*10)/32768;
	 EL3174_Channel4_Alarm:=  EL3174_Channel4_value>(2.5*10)/32768;
    GVL.NumericOutput[101] := SHL(TO_DWORD(GVL.SystemFlags), 0) OR 
                              SHL(TO_DWORD(GVL.EthercatAliveFromMaster), 2) OR 
                              SHL(TO_DWORD(GVL.RemoteMasterAlive), 3) OR 
                              SHL(TO_DWORD(watchDog), 4) OR 
                              SHL(TO_DWORD(DataRefreshRequired), 5) OR
                              SHL(TO_DWORD(IsInitPhase), 6) OR 
							  SHL(TO_DWORD(EL3174_Channel1_Alarm), 7) OR 
							  SHL(TO_DWORD(EL3174_Channel2_Alarm), 8) OR 
							  SHL(TO_DWORD(EL3174_Channel3_Alarm), 9) OR 
							  SHL(TO_DWORD(EL3174_Channel4_Alarm), 10);
    GVL.NumericOutput[102] := SHL(TO_DWORD(GVL.GroupMaster[0]), 16) OR TO_DWORD(GVL.GroupMaster[1]);
    GVL.NumericOutput[103] := SHL(TO_DWORD(GVL.GroupMaster[2]), 16) OR TO_DWORD(GVL.GroupMaster[3]);

   // GVL.NumericOutput[100] := systemAlarms;
    GVL.NumericOutput[108] := UINT_TO_DWORD(GVL.GroupCapacity[0]);
    GVL.NumericOutput[109] := UINT_TO_DWORD(GVL.GroupCapacity[1]);
    GVL.NumericOutput[110] := UINT_TO_DWORD(GVL.GroupCapacity[2]);
    GVL.NumericOutput[111] := UINT_TO_DWORD(GVL.GroupCapacity[3]);
END_IF;
END_METHOD

END_FUNCTION_BLOCK

// ---- POU/DeviceManager.TcPOU
FUNCTION_BLOCK DeviceManager
VAR_INPUT
  DeviceIndex : INT;                          // Index of device (0-19)
  Reset : BOOL;                               // Reset polling state
  Command : INT;                              // Unused input (for compatibility)
END_VAR
VAR
  CANBusIndex : INT;                          // CAN bus number (1-3)
  DeviceOffset : INT;                         // Offset within bus (0-7)
  rxData : RxData;                            // Received CAN data
  txData : TxData;                            // Transmitted CAN data
  PollCounter : INT := 0;                     // Counter for polling interval
  ResponseTrigger : R_TRIG;                   // Trigger for response detection
  LastExpectedCommand : UINT;                 // Last command sent
  InitDone : BOOL;                            // Initialization complete flag
  CommandIndex : INT := 0;                    // Current command index during init
  DeviceChanged : BOOL;                       // Flag for detected device change
  
  i : INT;                                    // Loop variable
  currentTime : TIME;                         // Current PLC time
  rawValue : UINT;                            // 2-byte value from CAN response
  statusLow : BYTE;                           // Low byte of SYSTEM_STATUS
  factorNibble : UINT;                        // Factor nibble from scaling-factor fields
  serialMismatch : BOOL;                      // Flag for serial number mismatch
	watchDog: INT;
END_VAR
VAR CONSTANT
  PollInterval : INT := 3;                    // Poll every 3 cycles (~30ms at 10ms cycle)
  ReadCommands : ARRAY[0..13] OF UINT := [GVL_Constant.CMD_READ_VIN,
                                          GVL_Constant.CMD_READ_VOUT,
                                          GVL_Constant.CMD_READ_IOUT,
                                          GVL_Constant.CMD_SCALING_FACTOR,
                                          GVL_Constant.CMD_SYSTEM_STATUS,
                                          GVL_Constant.CMD_READ_TEMPERATURE_1,
                                          GVL_Constant.CMD_READ_FAN_SPEED1,
                                          GVL_Constant.CMD_READ_FAN_SPEED2,
                                          GVL_Constant.CMD_FAULT_STATUS,
                                          GVL_Constant.CMD_OPERATION,
                                          GVL_Constant.CMD_DIRECTION_CTRL,
                                          GVL_Constant.CMD_REVERSE_VOUT_SET,
                                          GVL_Constant.CMD_REVERSE_IOUT_SET];
  ReadCommandCount : INT := 13;               // Number of read commands
  TotalInitCommands : INT := 22;              // Total commands in init (13 read + 9 MFR)
END_VAR

METHOD Poll : BOOL
VAR
  pollIntervalLocal : INT;
END_VAR
(** Initialize CAN bus and device offset mapping based on DeviceIndex (0-19) **)
CASE DeviceIndex OF
  0..3: CANBusIndex := 1; DeviceOffset := DeviceIndex; (** Map devices 0-3 to CAN Bus 1, offset 0-3 **)
  4..11: CANBusIndex := 2; DeviceOffset := DeviceIndex - 4; (** Map devices 4-11 to CAN Bus 2, offset 0-7 **)
  12..19: CANBusIndex := 3; DeviceOffset := DeviceIndex - 12; (** Map devices 12-19 to CAN Bus 3, offset 0-7 **)
  ELSE Poll := FALSE; RETURN; (** Disable polling and exit for invalid DeviceIndex **)
END_CASE;

(** Assign receive (rxData) and transmit (txData) structures based on CAN bus **)
CASE CANBusIndex OF
  1: rxData := GVL.Bus1_Devices_Rx[DeviceOffset]; txData := GVL.Bus1_Devices[DeviceOffset]; (** Use Bus 1 data structures **)
  2: rxData := GVL.Bus2_Devices_Rx[DeviceOffset]; txData := GVL.Bus2_Devices[DeviceOffset]; (** Use Bus 2 data structures **)
  3: rxData := GVL.Bus3_Devices_Rx[DeviceOffset]; txData := GVL.Bus3_Devices[DeviceOffset]; (** Use Bus 3 data structures **)
END_CASE;

currentTime := TIME(); (** Capture current time for timeout and update tracking **)

(** Reset all polling and initialization state if Reset is triggered **)
IF Reset THEN
  PollCounter := 0; (** Reset polling counter **)
  InitDone := FALSE; (** Mark initialization as not complete **)
  CommandIndex := 0; (** Reset command index to start of sequence **)
  DeviceChanged := FALSE; (** Clear device change flag **)
  LastExpectedCommand := 0; (** Clear last expected command **)
  GVL.ReadCommandIndex[DeviceIndex] := 0; (** Reset read command index **)
  // Remove persistent init flag since we're not using persistent storage
END_IF;

(** Check if polling pause has timed out **)
IF GVL.PollingPaused[DeviceIndex] AND GVL.PollingPauseTimeout[DeviceIndex].Q THEN
  GVL.PollingPaused[DeviceIndex] := FALSE; (** Resume polling after timeout **)
  GVL.PollingPauseTimeout[DeviceIndex](IN := FALSE); (** Stop timeout **)
END_IF;

PollCounter := PollCounter + 1; (** Increment polling counter **)

pollIntervalLocal := PollInterval;
IF DeviceIndex <= 3 THEN
  pollIntervalLocal := 5; (** DPU minimum request period is 50 ms; task loop is 10 ms **)
END_IF;

(** Trigger polling action if counter reaches interval and polling is not paused **)
IF PollCounter >= pollIntervalLocal AND NOT GVL.PollingPaused[DeviceIndex] THEN
  PollCounter := 0; (** Reset counter for next interval **)
  IF NOT InitDone OR DeviceChanged THEN (** Enter initialization or reinitialization phase **)
    IF CommandIndex < TotalInitCommands THEN (** Continue if more commands to process **)
      IF CommandIndex < ReadCommandCount THEN
        LastExpectedCommand := ReadCommands[CommandIndex]; (** Use operational commands first **)
        IF DeviceIndex <= 3 AND (LastExpectedCommand = GVL_Constant.CMD_SCALING_FACTOR OR LastExpectedCommand = GVL_Constant.CMD_SYSTEM_STATUS) THEN
          LastExpectedCommand := GVL_Constant.CMD_READ_VIN; (** DPU devices do not use BIC-only factor/status commands **)
        END_IF;
      ELSE
        // Ensure ID commands are polled first
        CASE CommandIndex - ReadCommandCount OF
          0: LastExpectedCommand := GVL_Constant.CMD_MFR_ID_B0B5; (** Poll ID bytes 0-5 **)
          1: LastExpectedCommand := GVL_Constant.CMD_MFR_ID_B6B11; (** Poll ID bytes 6-11 **)
          2: LastExpectedCommand := GVL_Constant.CMD_MFR_MODEL_B0B5; (** Poll model bytes 0-5 **)
          3: LastExpectedCommand := GVL_Constant.CMD_MFR_MODEL_B6B11; (** Poll model bytes 6-11 **)
          4: LastExpectedCommand := GVL_Constant.CMD_MFR_REVISION_B0B5; (** Poll revision bytes 0-5 **)
          5: LastExpectedCommand := GVL_Constant.CMD_MFR_LOCATION_B0B2; (** Poll location bytes 0-2 **)
          6: LastExpectedCommand := GVL_Constant.CMD_MFR_DATE_B0B5; (** Poll date bytes 0-5 **)
          7: LastExpectedCommand := GVL_Constant.CMD_MFR_SERIAL_B0B5; (** Poll serial bytes 0-5 **)
          8: LastExpectedCommand := GVL_Constant.CMD_MFR_SERIAL_B6B11; (** Poll serial bytes 6-11 **)
          ELSE LastExpectedCommand := GVL_Constant.MfrCommands[CommandIndex - ReadCommandCount]; (** Fallback to original MfrCommands **)
        END_CASE;
      END_IF;
      txData.Command := UINT_TO_INT(LastExpectedCommand); (** Assign command **)
      txData.Data[0] := 0; (** No data for read commands **)
      txData.Data[1] := 0;
      txData.Data[2] := 0;
      txData.Data[3] := 0;
    ELSE
      InitDone := TRUE; (** Mark initialization complete **)
      DeviceChanged := FALSE; (** Clear change flag **)
      Poll := FALSE; (** Stop polling **)
      RETURN; (** Exit method **)
    END_IF;
  ELSE (** Normal operation phase after initialization **)
    LastExpectedCommand := ReadCommands[GVL.ReadCommandIndex[DeviceIndex]]; (** Use next operational command **)
    IF DeviceIndex <= 3 AND (LastExpectedCommand = GVL_Constant.CMD_SCALING_FACTOR OR LastExpectedCommand = GVL_Constant.CMD_SYSTEM_STATUS) THEN
      LastExpectedCommand := GVL_Constant.CMD_READ_VIN; (** DPU devices do not use BIC-only factor/status commands **)
    END_IF;
    IF GVL.ReadCommandIndex[DeviceIndex] = ReadCommandCount - 1 THEN (** Last command in cycle **)
      LastExpectedCommand := GVL_Constant.CMD_MFR_SERIAL_B6B11; (** Poll serial command periodically **)
    END_IF;
    txData.Command := UINT_TO_INT(LastExpectedCommand); (** Assign command **)
    txData.Data[0] := 0; (** No data for read commands **)
    txData.Data[1] := 0;
    txData.Data[2] := 0;
    txData.Data[3] := 0;
    GVL.ReadCommandIndex[DeviceIndex] := GVL.ReadCommandIndex[DeviceIndex] + 1; (** Move to next command **)
    IF GVL.ReadCommandIndex[DeviceIndex] >= ReadCommandCount THEN
      GVL.ReadCommandIndex[DeviceIndex] := 0; (** Cycle back if at end **)
    END_IF;
  END_IF;

  (** Send command to appropriate CAN bus **)
  CASE CANBusIndex OF
    1: GVL.Bus1_Devices[DeviceOffset] := txData; (** Send command to Bus 1 **)
    2: GVL.Bus2_Devices[DeviceOffset] := txData; (** Send to Bus 2 **)
    3: GVL.Bus3_Devices[DeviceOffset] := txData; (** Send to Bus 3 **)
  END_CASE;
  Poll := TRUE; (** Signal polling action **)
END_IF;

(** Check if received command matches the last sent command to trigger response processing **)
ResponseTrigger(CLK := (rxData.Command = UINT_TO_INT(LastExpectedCommand)));
IF ResponseTrigger.Q THEN (** Response received and matches expected command **)
  rawValue := rxData.Data[0] + SHL(rxData.Data[1], 8); (** Combine first two bytes into a 16-bit value **)
  CASE LastExpectedCommand OF

	GVL_Constant.CMD_READ_VIN: GVL.Vin[DeviceIndex] := rawValue; (** Update VIN **)
	GVL_Constant.CMD_READ_VOUT: GVL.Vout[DeviceIndex] := rawValue; (** Update VOUT **)
	GVL_Constant.CMD_READ_IOUT:  GVL.Iout[DeviceIndex] := rawValue; (** Default to raw value **)
    GVL_Constant.CMD_SCALING_FACTOR:
      GVL.VoutScale[DeviceIndex] := rawValue; (** Low nibble=VOUT factor, high nibble=IOUT factor, byte1 holds VIN/FAN factors **)
      GVL.VinScale[DeviceIndex] := SHR(rawValue, 8);
    GVL_Constant.CMD_SYSTEM_STATUS:
      statusLow := UINT_TO_BYTE(rawValue AND 16#00FF);
      GVL.Ms[DeviceIndex] := (statusLow AND 16#01) <> 0;           (** Bit0 M/S **)
      GVL.DcOk[DeviceIndex] := (statusLow AND 16#02) <> 0;         (** Bit1 DC_OK **)
      GVL.PfcOk[DeviceIndex] := (statusLow AND 16#04) <> 0;        (** Bit2 PFC_OK **)
      GVL.AdlOn[DeviceIndex] := (statusLow AND 16#08) <> 0;        (** Bit3 ADL_ON **)
      GVL.InitialState[DeviceIndex] := (statusLow AND 16#10) <> 0; (** Bit4 INITIAL_STATE **)
      GVL.Eeper[DeviceIndex] := (statusLow AND 16#20) <> 0;        (** Bit5 EEPER **)
    GVL_Constant.CMD_READ_TEMPERATURE_1: GVL.Temperature[DeviceIndex] := rawValue; (** Update temperature **)
    GVL_Constant.CMD_READ_FAN_SPEED1: GVL.FanSpeed1[DeviceIndex] := rawValue; (** Update fan speed 1 **)
    GVL_Constant.CMD_READ_FAN_SPEED2: GVL.FanSpeed2[DeviceIndex] := rawValue; (** Update fan speed 2 **)
    GVL_Constant.CMD_FAULT_STATUS: GVL.FaultStatus[DeviceIndex] := rawValue; (** Update fault status **)
    GVL_Constant.CMD_OPERATION: GVL.OperationOn[DeviceIndex] := (rawValue > 0); (** Update operation state **)
    GVL_Constant.CMD_VOUT_SET:
      IF DeviceIndex <= 3 THEN
        GVL.VoutSetpoint[DeviceIndex] := UINT_TO_REAL(rawValue) / 10.0;   (** DPU F=0.1 **)
      ELSE
        factorNibble := GVL.VoutScale[DeviceIndex] AND 16#000F;
        CASE factorNibble OF
          16#4: GVL.VoutSetpoint[DeviceIndex] := UINT_TO_REAL(rawValue) * 0.001;
          16#5: GVL.VoutSetpoint[DeviceIndex] := UINT_TO_REAL(rawValue) * 0.01;
          16#6: GVL.VoutSetpoint[DeviceIndex] := UINT_TO_REAL(rawValue) * 0.1;
          16#7: GVL.VoutSetpoint[DeviceIndex] := UINT_TO_REAL(rawValue);
          16#8: GVL.VoutSetpoint[DeviceIndex] := UINT_TO_REAL(rawValue) * 10.0;
          16#9: GVL.VoutSetpoint[DeviceIndex] := UINT_TO_REAL(rawValue) * 100.0;
          ELSE GVL.VoutSetpoint[DeviceIndex] := UINT_TO_REAL(rawValue) * 0.01;
        END_CASE;
      END_IF;
    GVL_Constant.CMD_IOUT_SET:
      IF DeviceIndex <= 3 THEN
        GVL.IoutSetpoint[DeviceIndex] := UINT_TO_REAL(rawValue) / 10.0;   (** DPU F=0.1 **)
      ELSE
        factorNibble := SHR((GVL.VoutScale[DeviceIndex] AND 16#00F0), 4);
        CASE factorNibble OF
          16#4: GVL.IoutSetpoint[DeviceIndex] := UINT_TO_REAL(rawValue) * 0.001;
          16#5: GVL.IoutSetpoint[DeviceIndex] := UINT_TO_REAL(rawValue) * 0.01;
          16#6: GVL.IoutSetpoint[DeviceIndex] := UINT_TO_REAL(rawValue) * 0.1;
          16#7: GVL.IoutSetpoint[DeviceIndex] := UINT_TO_REAL(rawValue);
          16#8: GVL.IoutSetpoint[DeviceIndex] := UINT_TO_REAL(rawValue) * 10.0;
          16#9: GVL.IoutSetpoint[DeviceIndex] := UINT_TO_REAL(rawValue) * 100.0;
          ELSE GVL.IoutSetpoint[DeviceIndex] := UINT_TO_REAL(rawValue) * 0.01;
        END_CASE;
      END_IF;

    GVL_Constant.CMD_MFR_ID_B0B5: (** Manufacturer ID bytes 0-5 **)
      FOR i := 0 TO 5 DO
        GVL.MfrSerialPersistent[DeviceIndex][i] := rxData.Data[i]; (** Store first 6 bytes in non-persistent array **)
      END_FOR;
    GVL_Constant.CMD_MFR_ID_B6B11: (** Manufacturer ID bytes 6-11 **)
      FOR i := 0 TO 5 DO
        GVL.MfrSerialPersistent[DeviceIndex][6 + i] := rxData.Data[i]; (** Store next 6 bytes in non-persistent array **)
      END_FOR;
    GVL_Constant.CMD_MFR_MODEL_B0B5: (** Manufacturer model bytes 0-5 **)
      FOR i := 0 TO 5 DO
        GVL.MfrSerialPersistent[DeviceIndex][12 + i] := rxData.Data[i]; (** Store model bytes 12-17 **)
      END_FOR;
    GVL_Constant.CMD_MFR_MODEL_B6B11: (** Manufacturer model bytes 6-11 **)
      FOR i := 0 TO 5 DO
        GVL.MfrSerialPersistent[DeviceIndex][18 + i] := rxData.Data[i]; (** Store model bytes 18-23 **)
      END_FOR;
    GVL_Constant.CMD_MFR_REVISION_B0B5: (** Manufacturer revision bytes 0-5 **)
      FOR i := 0 TO 5 DO
        GVL.MfrSerialPersistent[DeviceIndex][24 + i] := rxData.Data[i]; (** Store revision bytes 24-29 **)
      END_FOR;
    GVL_Constant.CMD_MFR_LOCATION_B0B2: (** Manufacturer location bytes 0-2 **)
      FOR i := 0 TO 2 DO
        GVL.MfrSerialPersistent[DeviceIndex][30 + i] := rxData.Data[i]; (** Store location bytes 30-32 **)
      END_FOR;
    GVL_Constant.CMD_MFR_DATE_B0B5: (** Manufacturer date bytes 0-5 **)
      FOR i := 0 TO 5 DO
        GVL.MfrSerialPersistent[DeviceIndex][33 + i] := rxData.Data[i]; (** Store date bytes 33-38 **)
      END_FOR;
    GVL_Constant.CMD_MFR_SERIAL_B0B5: (** Manufacturer serial bytes 0-5 **)
      FOR i := 0 TO 5 DO
        GVL.MfrSerialPersistent[DeviceIndex][39 + i] := rxData.Data[i]; (** Store serial bytes 39-44 **)
      END_FOR;
    GVL_Constant.CMD_MFR_SERIAL_B6B11: (** Manufacturer serial bytes 6-11 **)
      FOR i := 0 TO 5 DO
        GVL.MfrSerialPersistent[DeviceIndex][45 + i] := rxData.Data[i]; (** Store serial bytes 45-50 **)
        IF GVL.MfrSerialPersistent[DeviceIndex][39 + i] <> rxData.Data[i] THEN (** Check for serial mismatch **)
          serialMismatch := TRUE;
        END_IF;
      END_FOR;
      IF serialMismatch AND InitDone THEN (** Trigger reinitialization if mismatch after init **)
        DeviceChanged := TRUE;
        CommandIndex := 0;
        InitDone := FALSE;
      END_IF;
  END_CASE;

  GVL.CommTimeouts[DeviceIndex] := 0; (** Reset timeout counter on successful response **)
  GVL.SuccessCounts[DeviceIndex] := GVL.SuccessCounts[DeviceIndex] + 1; (** Increment success count **)
  IF GVL.SuccessCounts[DeviceIndex] >= GVL_Constant.MINSUCCESSCLEAR THEN (** Clear faults after sufficient successes **)
    GVL.CommFault[DeviceIndex] := FALSE;
    GVL.FaultLevel[DeviceIndex] := 0;
    GVL.RecoveryPending[DeviceIndex] := FALSE;
    GVL.SuccessCounts[DeviceIndex] := GVL_Constant.MINSUCCESSCLEAR;
  END_IF;
  GVL.LastUpdateTime[DeviceIndex] := currentTime; (** Update last successful time **)
  GVL.DataValid[DeviceIndex] := TRUE; (** Mark data as valid **)
  Poll := TRUE; (** Continue polling **)

  IF NOT InitDone THEN (** Advance command index during initialization **)
    CommandIndex := CommandIndex + 1;
  END_IF;
ELSE (** No response received **)
  IF PollCounter = 0 AND LastExpectedCommand <> 0 THEN (** Check timeout at interval start **)
    IF (currentTime - GVL.LastUpdateTime[DeviceIndex]) > GVL_Constant.MAXCOMMSTALE THEN
      GVL.CommTimeouts[DeviceIndex] := GVL.CommTimeouts[DeviceIndex] + pollIntervalLocal; (** Increment timeout **)
      GVL.SuccessCounts[DeviceIndex] := 0; (** Reset success count on timeout **)
      IF GVL.CommTimeouts[DeviceIndex] >= GVL_Constant.MAXCOMMTIMEOUT THEN (** Trigger fault if timeout exceeds **)
        GVL.CommFault[DeviceIndex] := TRUE;
        GVL.RecoveryPending[DeviceIndex] := TRUE;
        GVL.FaultLevel[DeviceIndex] := 1;
      END_IF;
      IF NOT InitDone THEN (** Advance command on timeout during init **)
        CommandIndex := CommandIndex + 1;
      END_IF;
    END_IF;
  END_IF;
END_IF;

(** Invalidate data if stale **)
IF (currentTime - GVL.LastUpdateTime[DeviceIndex]) > GVL_Constant.MAXCOMMSTALE THEN
  GVL.DataValid[DeviceIndex] := FALSE;
END_IF;

(** Ensure full initialization on first run **)
IF GVL.FirstRun AND NOT InitDone THEN
  CommandIndex := 0; (** Reset to start initialization **)
END_IF;
END_METHOD

METHOD WriteDLC3 : BOOL
VAR_INPUT
  DeviceIndex : INT;                       (* Device index *)
  WriteCommandIndex : UINT;                (* Command to send *)
  Data : BYTE;                             (* Single-byte data *)
END_VAR
VAR
  txDataLocal : TxData;                    (* Transmit data structure *)
END_VAR

CASE DeviceIndex OF
  0..3: CANBusIndex := 1; DeviceOffset := DeviceIndex;
  4..11: CANBusIndex := 2; DeviceOffset := DeviceIndex - 4;
  12..19: CANBusIndex := 3; DeviceOffset := DeviceIndex - 12;
  ELSE WriteDLC3 := FALSE; RETURN;
END_CASE;

txDataLocal.Command := UINT_TO_INT(WriteCommandIndex);
txDataLocal.Data[0] := Data;
txDataLocal.Data[1] := 0;
txDataLocal.Data[2] := 0;
txDataLocal.Data[3] := 0;

CASE CANBusIndex OF
  1: GVL.Bus1_Devices_DLC3[DeviceOffset] := txDataLocal; WriteDLC3 := TRUE;
  2: GVL.Bus2_Devices_DLC3[DeviceOffset] := txDataLocal; WriteDLC3 := TRUE;
  3: GVL.Bus3_Devices_DLC3[DeviceOffset] := txDataLocal; WriteDLC3 := TRUE;
END_CASE;

IF WriteCommandIndex = GVL_Constant.CMD_OPERATION THEN
  GVL.OperationOn[DeviceIndex] := FALSE; (* Reset to avoid latching *)
  GVL.OperationOn[DeviceIndex] := (Data > 0) AND NOT GVL.Standby[DeviceIndex];
ELSIF WriteCommandIndex = GVL_Constant.CMD_DIRECTION_CTRL THEN
  GVL.Direction[DeviceIndex] := (Data > 0);
END_IF;
END_METHOD

METHOD WriteDLC4 : BOOL
VAR_INPUT
  DeviceIndex : INT;                       (** Device index **)
  WriteCommandIndex : INT;                 (** Command to send **)
  Data : UINT;                             (** 2-byte data **)
END_VAR
VAR
  txDataLocal : TxData;                    (** Transmit data structure **)
END_VAR

         
(** Map DeviceIndex to CAN bus and offset **)
CASE DeviceIndex OF
  0..3: CANBusIndex := 1; DeviceOffset := DeviceIndex; (** Devices 0-3 map to Bus 1, offset 0-3 **)
  4..11: CANBusIndex := 2; DeviceOffset := DeviceIndex - 4; (** Devices 4-11 map to Bus 2, offset 0-7 **)
  12..19: CANBusIndex := 3; DeviceOffset := DeviceIndex - 12; (** Devices 12-19 map to Bus 3, offset 0-7 **)
  ELSE WriteDLC4 := FALSE; RETURN; (** Invalid DeviceIndex, exit **)
END_CASE;


  (** Output enabled, proceed with normal data **)
  txDataLocal.Command := WriteCommandIndex;
  txDataLocal.Data[0] := UINT_TO_BYTE(Data AND 16#FF); (** Low byte **)
  txDataLocal.Data[1] := UINT_TO_BYTE(SHR(Data, 8)); (** High byte **)
  txDataLocal.Data[2] := 0; (** Clear unused bytes **)
  txDataLocal.Data[3] := 0;

(** Write to appropriate CAN bus output **)
CASE CANBusIndex OF
  1: 
    IF DeviceOffset >= 0 AND DeviceOffset <= 3 THEN
      GVL.Bus1_Devices_DLC4[DeviceOffset] := txDataLocal; (** Update Bus 1 DLC4 for devices 0-3 **)
      WriteDLC4 := TRUE;
    ELSE
      WriteDLC4 := FALSE; (** Invalid offset for Bus 1 **)
    END_IF;
  2: 
    IF DeviceOffset >= 0 AND DeviceOffset <= 7 THEN
      GVL.Bus2_Devices_DLC4[DeviceOffset] := txDataLocal; (** Update Bus 2 DLC4 **)
      WriteDLC4 := TRUE;
    ELSE
      WriteDLC4 := FALSE; (** Invalid offset for Bus 2 **)
    END_IF;
  3: 
    IF DeviceOffset >= 0 AND DeviceOffset <= 7 THEN
      GVL.Bus3_Devices_DLC4[DeviceOffset] := txDataLocal; (** Update Bus 3 DLC4 **)
      WriteDLC4 := TRUE;
    ELSE
      WriteDLC4 := FALSE; (** Invalid offset for Bus 3 **)
    END_IF;
END_CASE;

(** Update GVL variables based on command **)
IF WriteDLC4 THEN
  IF WriteCommandIndex = GVL_Constant.CMD_VOUT_SET THEN
    GVL.VoutSetpoint[DeviceIndex] := UINT_TO_REAL(Data); (** Update Vout setpoint **)
  ELSIF WriteCommandIndex = GVL_Constant.CMD_IOUT_SET THEN
    GVL.IoutSetpoint[DeviceIndex] := UINT_TO_REAL(Data); (** Update Iout setpoint **)
  ELSIF WriteCommandIndex = GVL_Constant.CMD_REVERSE_VOUT_SET THEN
    GVL.VoutSetRev[DeviceIndex] := UINT_TO_REAL(Data); (** Update reverse Vout **)
  ELSIF WriteCommandIndex = GVL_Constant.CMD_REVERSE_IOUT_SET THEN
    GVL.IoutSetRev[DeviceIndex] := UINT_TO_REAL(Data);(** Update reverse Iout **)
  END_IF;
END_IF;
END_METHOD

END_FUNCTION_BLOCK

// ---- POU/SafetyMgr.TcPOU
FUNCTION_BLOCK SafetyMgr
VAR
  OrangeFault : BOOL;                         // Orange-level fault detected
  RedFault : BOOL;                            // Red-level fault detected
  AlarmBits : UINT;                           // Bitmask of alarmed devices
  RecoveryTrigger : BOOL;                     // Trigger for recovery attempt
  Watchdog : TON;                             // EtherCAT watchdog timer
  AllOutputsOff : BOOL;                       // All outputs are off
  ShutdownActive : ARRAY[0..19] OF BOOL;      // Shutdown in progress per device
  FastOffActive : ARRAY[0..19] OF BOOL;       // Fast off in progress per device
  AnyOutputOn : BOOL;                         // Any output is on
  EStopTimer : TON;                           // E-Stop delay timer
  RedStopTimer : TON;                         // Red Stop delay timer
  OrangeStopTimer : TON;                      // Orange Stop delay timer
END_VAR

// Check if a device is safe to operate
METHOD IsDeviceSafe : BOOL
VAR_INPUT
  DeviceIndex : INT;                          // Device to check
END_VAR
IsDeviceSafe := DeviceIndex >= 0 AND DeviceIndex <= 19 AND GVL.FaultLevel[DeviceIndex] = 0 AND NOT ShutdownActive[DeviceIndex];
GVL.SafetyOK[DeviceIndex] := IsDeviceSafe;    // Update safety status
END_METHOD

// Update safety conditions and system state, handling E-Stop, Red/Orange Stops, and communication faults
METHOD UpdateSafety
VAR
  devIdx : INT;            (* Device index for iteration, 0-19 *)
  anyEStop : BOOL;         (* Aggregate E-Stop state across all devices *)
  anyRedStop : BOOL;       (* Aggregate Red Stop state across all devices *)
  anyOrangeStop : BOOL;    (* Aggregate Orange Stop state across all devices *)
  systemSafe : BOOL;       (* System-wide safety condition, false if alarms active *)
END_VAR
(* Initialize aggregate safety flags *)
anyEStop := FALSE;
anyRedStop := FALSE;
anyOrangeStop := FALSE;

// Aggregate device-level safety conditions
FOR devIdx := 0 TO 19 DO
  anyEStop := anyEStop OR GVL.EStop[devIdx];         (* Check device E-Stop *)
  anyRedStop := anyRedStop OR GVL.RedStop[devIdx];   (* Check device Red Stop *)
  anyOrangeStop := anyOrangeStop OR GVL.OrangeStop[devIdx]; (* Check device Orange Stop *)
END_FOR;

// Update system state based on aggregated conditions
IF anyEStop THEN
  GVL.SystemState := 3; // E-Stop state, highest priority
ELSIF anyRedStop THEN
  GVL.SystemState := 2; // Red Stop state
ELSIF anyOrangeStop THEN
  GVL.SystemState := 1; // Orange Stop state
ELSE
  GVL.SystemState := 0; // Normal state, all clear
END_IF;

// Update SafetyOK per device: safe if no E-Stop, Red, or Orange Stop
FOR devIdx := 0 TO 19 DO
  GVL.SafetyOK[devIdx] := NOT (GVL.EStop[devIdx] OR GVL.RedStop[devIdx] OR GVL.OrangeStop[devIdx]);
END_FOR;

// Check system-wide alarms for safety condition
IF GVL.AlarmStatus <> 0 THEN // Non-zero AlarmStatus indicates active alarms
  systemSafe := FALSE;
ELSE
  systemSafe := TRUE;
END_IF;

// Apply system-wide safety and device-specific faults to shutdown
FOR devIdx := 0 TO 19 DO
  GVL.SafetyShutdown[devIdx] := NOT systemSafe OR GVL.CommFault[devIdx] OR GVL.TemperatureFaultHigh[devIdx];
END_FOR;

// Disable outputs for devices in shutdown
FOR devIdx := 0 TO 19 DO
  IF GVL.SafetyShutdown[devIdx] THEN
    GVL.OutputOn[devIdx] := FALSE; // Disable output on shutdown
  END_IF;
END_FOR;

// Handle recovery: clear RecoveryPending if SafetyRecovery and device is safe
FOR devIdx := 0 TO 19 DO
  IF GVL.SafetyRecovery AND GVL.SafetyOK[devIdx] THEN
    GVL.RecoveryPending[devIdx] := FALSE;
  END_IF;
END_FOR;

// Update fault level per device based on stop conditions
FOR devIdx := 0 TO 19 DO
  IF GVL.EStop[devIdx] THEN
    GVL.FaultLevel[devIdx] := 2; // Red fault level
  ELSIF GVL.OrangeStop[devIdx] THEN
    GVL.FaultLevel[devIdx] := 1; // Orange fault level
  ELSE
    GVL.FaultLevel[devIdx] := 0; // No fault
  END_IF;
END_FOR;

// Update communication faults and polling status
FOR devIdx := 0 TO 19 DO
  GVL.CommFault[devIdx] := GVL.CommTimeouts[devIdx] > GVL_constant.MAXCOMMTIMEOUT; (* Fixed: MAXCOMMTIMEOUT *)
  GVL.PollingPaused[devIdx] := GVL.CommFault[devIdx] AND NOT GVL.DataValid[devIdx]; (* Pause polling if fault and stale *)
  GVL.RecoveryPending[devIdx] := GVL.RecoveryPending[devIdx] OR (GVL.FaultLevel[devIdx] > 0); (* Set pending if faulted *)
END_FOR;
END_METHOD

END_FUNCTION_BLOCK

// ---- POU/GroupManager.TcPOU

FUNCTION_BLOCK GroupManager
VAR
  i : INT;                                    // Loop variable for devices
  groupIdx : INT;                             // Group index
  groupBase : INT;                            // Base device index for group
	devIdx: INT;
END_VAR

FOR devIdx := 0 TO 19 DO
  IF devIdx < 4 THEN
    GVL.GroupMembership[devIdx] := -1; (** Devices 0-3 not in groups **)
  ELSIF devIdx >= 4 AND devIdx <= 7 THEN
    GVL.GroupMembership[devIdx] := 0; (** Group 0: devices 4-7 **)
  ELSIF devIdx >= 8 AND devIdx <= 11 THEN
    GVL.GroupMembership[devIdx] := 1; (** Group 1: devices 8-11 **)
  ELSIF devIdx >= 12 AND devIdx <= 15 THEN
    GVL.GroupMembership[devIdx] := 2; (** Group 2: devices 12-15 **)
  ELSIF devIdx >= 16 AND devIdx <= 19 THEN
    GVL.GroupMembership[devIdx] := 3; (** Group 3: devices 16-19 **)
  END_IF;
END_FOR;

METHOD UpdateGroupCapacity
VAR
  activeDevices : INT;                        (** Count of active devices in group **)
  devIdx : INT;                              (** Device index **)
  groupBase : INT;                           (** Base index for group devices **)
  opCount : UINT;                            (** Count of devices with OperationOn **)
  outCount : UINT;                           (** Count of devices with OutputOn **)
END_VAR

FOR groupIdx := 0 TO 3 DO
  groupBase := groupIdx * 4 + 4;              (** Groups: 0=4-7, 1=8-11, 2=12-15, 3=16-19 **)
  activeDevices := 0;
  opCount := 0;
  outCount := 0;
  GVL.GroupCapacity[groupIdx] := 0;

  (** Calculate active devices based on input voltage feedback **)
  FOR devIdx := groupBase TO groupBase + 3 DO
    IF devIdx <= 19 THEN
      IF GVL.Vin[devIdx] > 100 THEN
        activeDevices := activeDevices + 1;
      END_IF;
      IF GVL.OperationOn[devIdx] THEN
        opCount := opCount + 1;
      END_IF;
      IF GVL.OutputOn[devIdx] THEN
        outCount := outCount + 1;
      END_IF;
    END_IF;
  END_FOR;
  GVL.GroupCapacity[groupIdx] := activeDevices * GVL_Constant.IoutMax; (** 75A per device **)

  (** Update group status and alarms **)
  IF GVL.GroupMaster[groupIdx] >= 0 AND GVL.GroupMaster[groupIdx] <= 19 THEN
    GVL.NumericOutput[104 + groupIdx] := SHL(TO_DWORD(outCount), 16) OR TO_DWORD(opCount);
    IF opCount < 4 THEN
      GVL.SystemAlarms := DWORD_TO_UINT(GVL.SystemAlarms OR SHL(TO_DWORD(1), groupIdx));
    END_IF;
  ELSE
    GVL.NumericOutput[104 + groupIdx] := 0;
    GVL.GroupCapacity[groupIdx] := 0;
    GVL.SystemAlarms := DWORD_TO_UINT(GVL.SystemAlarms OR SHL(TO_DWORD(1), groupIdx));
  END_IF;
END_FOR;
END_METHOD

METHOD UpdateGroupMasters
VAR
  oldMaster : INT;                            (** Previous master index **)
  i : INT;                                    (** Loop variable for devices **)
  groupBase : INT;                           (** Base index for group devices **)
END_VAR

FOR groupIdx := 0 TO 3 DO
  groupBase := groupIdx * 4 + 4;              (** Groups: 0=4-7, 1=8-11, 2=12-15, 3=16-19 **)
  oldMaster := GVL.GroupMaster[groupIdx];
  GVL.GroupMaster[groupIdx] := -1;

  (** Retain current master if still healthy **)
  IF oldMaster >= groupBase AND oldMaster <= groupBase + 3 AND
     GVL.Vin[oldMaster] > 100 AND NOT GVL.CommFault[oldMaster] THEN
    GVL.GroupMaster[groupIdx] := oldMaster;
  ELSE
    (** Select first active healthy unit by VIN **)
    FOR i := groupBase TO groupBase + 3 DO
      IF i <= 19 AND GVL.Vin[i] > 100 AND NOT GVL.CommFault[i] THEN
        GVL.GroupMaster[groupIdx] := i;
        EXIT;
      END_IF;
    END_FOR;

    (** Final fallback for compatibility: base unit in group **)
    IF GVL.GroupMaster[groupIdx] = -1 AND groupBase <= 19 THEN
      GVL.GroupMaster[groupIdx] := groupBase;
    END_IF;
  END_IF;

  (** Set fault code if master changed **)
  IF oldMaster <> GVL.GroupMaster[groupIdx] AND GVL.GroupMaster[groupIdx] >= 0 THEN
    GVL.FaultStatus[GVL.GroupMaster[groupIdx]] := 8; (** Fault code 8 = master changed **)
  END_IF;
END_FOR;
END_METHOD

END_FUNCTION_BLOCK

// ---- POU/SetpointTest.TcPOU

(* ============================================================
   SetpointTest  –  TEMPORARY TEST PROGRAM
   Purpose:
     Inject group setpoints via GVL.TempGroupInput without
     touching live EtherCAT master inputs (GVL.NumericInput).

   Usage:
     1. Set GVL.UseTempGroupInputs := TRUE  to activate.
     2. Fill in the group parameters below (VoutTarget, IoutTarget,
        min/max limits, Flags) for whichever group you want to test.
     3. Call SetpointTest.Run() from Main or watch SetpointApplied.
     4. When finished, set GVL.UseTempGroupInputs := FALSE and
        clear GVL.TempGroupInput (Run() sets both automatically
        when Enable is set back to FALSE).

   REVERT NOTE:
     This POU together with GVL.UseTempGroupInputs / GVL.TempGroupInput
     and the ReadLimits conditional branch in EthercatManager must be
     removed once testing is complete.

   TempGroupInput layout (28 WORDs, groups 0-3 x 7 WORDs each):
     Offset 0  (group 0 base) : VoutSetpoint  (desired V * 100)
     Offset 1                 : IoutSetpoint  (desired A * 100)
     Offset 2                 : Flags         (bit 0=OutputOn, bit 1=OperationOn, bit 2=Voltage, bit 3=Current)
     Offset 3                 : VoutSetMin    (min V * 100)
     Offset 4                 : VoutSetMax    (max V * 100)
     Offset 5                 : IoutSetMin    (min A * 100)
     Offset 6                 : IoutSetMax    (max A * 100)
     Offset 7  (group 1 base) : same layout ...
   ============================================================ *)
PROGRAM SetpointTest
VAR
  Enable         : BOOL := FALSE;      (* Rising edge triggers injection; falling edge clears *)
  Enable_Prev    : BOOL := FALSE;      (* Previous value for edge detection *)

  EnableBus1Direct : BOOL := FALSE;    (* TRUE: directly drive devices 0..3 setpoints/flags *)
  Bus1DeviceMask   : BYTE := 16#0F;    (* bit0..bit3 select Bus1 devices to drive *)
  Bus1Direction    : BOOL := FALSE;    (* FALSE = AC->DC charge direction for DPU *)
  Bus1VoutTarget   : REAL := 28.0;     (* Direct voltage setpoint [V] for devices 0..3 *)
  Bus1IoutTarget   : REAL := 10.0;     (* Direct current setpoint [A] for devices 0..3 *)
  Bus1VoutSetMin   : REAL := 0.0;
  Bus1VoutSetMax   : REAL := 500.0;
  Bus1IoutSetMin   : REAL := 0.0;
  Bus1IoutSetMax   : REAL := 300.0;
  Bus1OutputOn     : BOOL := TRUE;
  Bus1OperationOn  : BOOL := TRUE;
  Bus1VoltageMode  : BOOL := TRUE;
  Bus1CurrentMode  : BOOL := FALSE;

  UseCommonAllGroups : BOOL := TRUE;   (* TRUE: push one shared profile to all 4 groups on enable *)
  CommonVoutTarget   : REAL := 28.0;   (* Shared voltage target [V] *)
  CommonIoutTarget   : REAL := 10.0;   (* Shared current target [A] *)
  CommonFlags        : WORD := 16#001A;(* bit1=OperationOn, bit3=Voltage, bit4=OutputOn *)
  CommonVoutSetMin   : REAL := 0.0;
  CommonVoutSetMax   : REAL := 500.0;
  CommonIoutSetMin   : REAL := 0.0;
  CommonIoutSetMax   : REAL := 300.0;

  (* Group 0 test parameters (indices 0-6 in TempGroupInput) *)
  G0_VoutTarget  : REAL := 28.0;       (* Desired voltage [V] – will be stored as WORD(value*100) *)
  G0_IoutTarget  : REAL := 10.0;       (* Desired current [A] – stored as WORD(value*100) *)
  G0_Flags       : WORD := 16#001A;    (* bit1=OperationOn, bit3=Voltage, bit4=OutputOn *)
  G0_VoutSetMin  : REAL := 0.0;
  G0_VoutSetMax  : REAL := 500.0;
  G0_IoutSetMin  : REAL := 0.0;
  G0_IoutSetMax  : REAL := 300.0;

  (* Group 1 test parameters (indices 7-13 in TempGroupInput) *)
  G1_VoutTarget  : REAL := 28.0;
  G1_IoutTarget  : REAL := 10.0;
  G1_Flags       : WORD := 16#001A;
  G1_VoutSetMin  : REAL := 0.0;
  G1_VoutSetMax  : REAL := 500.0;
  G1_IoutSetMin  : REAL := 0.0;
  G1_IoutSetMax  : REAL := 300.0;

  (* Group 2 test parameters (indices 14-20 in TempGroupInput) *)
  G2_VoutTarget  : REAL := 28.0;
  G2_IoutTarget  : REAL := 10.0;
  G2_Flags       : WORD := 16#001A;
  G2_VoutSetMin  : REAL := 0.0;
  G2_VoutSetMax  : REAL := 500.0;
  G2_IoutSetMin  : REAL := 0.0;
  G2_IoutSetMax  : REAL := 300.0;

  (* Group 3 test parameters (indices 21-27 in TempGroupInput) *)
  G3_VoutTarget  : REAL := 28.0;
  G3_IoutTarget  : REAL := 10.0;
  G3_Flags       : WORD := 16#001A;
  G3_VoutSetMin  : REAL := 0.0;
  G3_VoutSetMax  : REAL := 500.0;
  G3_IoutSetMin  : REAL := 0.0;
  G3_IoutSetMax  : REAL := 300.0;

  SetpointApplied : BOOL := FALSE;     (* TRUE while temp inputs are active *)
  busDev          : INT;
  bus1Applied     : BOOL := FALSE;
END_VAR


(* ---- While enabled: continuously refresh temp group inputs ---- *)
IF Enable THEN
  IF UseCommonAllGroups THEN
    G0_VoutTarget := CommonVoutTarget;
    G0_IoutTarget := CommonIoutTarget;
    G0_Flags := CommonFlags;
    G0_VoutSetMin := CommonVoutSetMin;
    G0_VoutSetMax := CommonVoutSetMax;
    G0_IoutSetMin := CommonIoutSetMin;
    G0_IoutSetMax := CommonIoutSetMax;

    G1_VoutTarget := CommonVoutTarget;
    G1_IoutTarget := CommonIoutTarget;
    G1_Flags := CommonFlags;
    G1_VoutSetMin := CommonVoutSetMin;
    G1_VoutSetMax := CommonVoutSetMax;
    G1_IoutSetMin := CommonIoutSetMin;
    G1_IoutSetMax := CommonIoutSetMax;

    G2_VoutTarget := CommonVoutTarget;
    G2_IoutTarget := CommonIoutTarget;
    G2_Flags := CommonFlags;
    G2_VoutSetMin := CommonVoutSetMin;
    G2_VoutSetMax := CommonVoutSetMax;
    G2_IoutSetMin := CommonIoutSetMin;
    G2_IoutSetMax := CommonIoutSetMax;

    G3_VoutTarget := CommonVoutTarget;
    G3_IoutTarget := CommonIoutTarget;
    G3_Flags := CommonFlags;
    G3_VoutSetMin := CommonVoutSetMin;
    G3_VoutSetMax := CommonVoutSetMax;
    G3_IoutSetMin := CommonIoutSetMin;
    G3_IoutSetMax := CommonIoutSetMax;
  END_IF;

  (* Group 0: TempGroupInput[0..6] *)
  GVL.TempGroupInput[0]  := REAL_TO_UINT(G0_VoutTarget * 100.0);
  GVL.TempGroupInput[1]  := REAL_TO_UINT(G0_IoutTarget * 100.0);
  GVL.TempGroupInput[2]  := G0_Flags;
  GVL.TempGroupInput[3]  := REAL_TO_UINT(G0_VoutSetMin * 100.0);
  GVL.TempGroupInput[4]  := REAL_TO_UINT(G0_VoutSetMax * 100.0);
  GVL.TempGroupInput[5]  := REAL_TO_UINT(G0_IoutSetMin * 100.0);
  GVL.TempGroupInput[6]  := REAL_TO_UINT(G0_IoutSetMax * 100.0);

  (* Group 1: TempGroupInput[7..13] *)
  GVL.TempGroupInput[7]  := REAL_TO_UINT(G1_VoutTarget * 100.0);
  GVL.TempGroupInput[8]  := REAL_TO_UINT(G1_IoutTarget * 100.0);
  GVL.TempGroupInput[9]  := G1_Flags;
  GVL.TempGroupInput[10] := REAL_TO_UINT(G1_VoutSetMin * 100.0);
  GVL.TempGroupInput[11] := REAL_TO_UINT(G1_VoutSetMax * 100.0);
  GVL.TempGroupInput[12] := REAL_TO_UINT(G1_IoutSetMin * 100.0);
  GVL.TempGroupInput[13] := REAL_TO_UINT(G1_IoutSetMax * 100.0);

  (* Group 2: TempGroupInput[14..20] *)
  GVL.TempGroupInput[14] := REAL_TO_UINT(G2_VoutTarget * 100.0);
  GVL.TempGroupInput[15] := REAL_TO_UINT(G2_IoutTarget * 100.0);
  GVL.TempGroupInput[16] := G2_Flags;
  GVL.TempGroupInput[17] := REAL_TO_UINT(G2_VoutSetMin * 100.0);
  GVL.TempGroupInput[18] := REAL_TO_UINT(G2_VoutSetMax * 100.0);
  GVL.TempGroupInput[19] := REAL_TO_UINT(G2_IoutSetMin * 100.0);
  GVL.TempGroupInput[20] := REAL_TO_UINT(G2_IoutSetMax * 100.0);

  (* Group 3: TempGroupInput[21..27] *)
  GVL.TempGroupInput[21] := REAL_TO_UINT(G3_VoutTarget * 100.0);
  GVL.TempGroupInput[22] := REAL_TO_UINT(G3_IoutTarget * 100.0);
  GVL.TempGroupInput[23] := G3_Flags;
  GVL.TempGroupInput[24] := REAL_TO_UINT(G3_VoutSetMin * 100.0);
  GVL.TempGroupInput[25] := REAL_TO_UINT(G3_VoutSetMax * 100.0);
  GVL.TempGroupInput[26] := REAL_TO_UINT(G3_IoutSetMin * 100.0);
  GVL.TempGroupInput[27] := REAL_TO_UINT(G3_IoutSetMax * 100.0);

  GVL.UseTempGroupInputs := TRUE;
  SetpointApplied := TRUE;
END_IF;

(* ---- Optional direct Bus1 (DPU) test path ---- *)
IF Enable AND EnableBus1Direct THEN
  GVL.UseTempBus1Direct := TRUE;
  FOR busDev := 0 TO 3 DO
    IF (Bus1DeviceMask AND SHL(16#01, busDev)) <> 0 THEN
      GVL.TempBus1VoutSetpoint[busDev] := REAL_TO_UINT(Bus1VoutTarget * 100.0);
      GVL.TempBus1IoutSetpoint[busDev] := REAL_TO_UINT(Bus1IoutTarget * 100.0);
      GVL.TempBus1Flags[busDev] := SEL(Bus1Direction, 16#0000, 16#0001)
                                OR SEL(Bus1OperationOn, 16#0000, 16#0002)
                                OR SEL(Bus1CurrentMode, 16#0000, 16#0004)
                                OR SEL(Bus1VoltageMode, 16#0000, 16#0008)
                                OR SEL(Bus1OutputOn, 16#0000, 16#0010);
      GVL.TempBus1VoutSetMin[busDev] := REAL_TO_UINT(Bus1VoutSetMin * 100.0);
      GVL.TempBus1VoutSetMax[busDev] := REAL_TO_UINT(Bus1VoutSetMax * 100.0);
      GVL.TempBus1IoutSetMin[busDev] := REAL_TO_UINT(Bus1IoutSetMin * 100.0);
      GVL.TempBus1IoutSetMax[busDev] := REAL_TO_UINT(Bus1IoutSetMax * 100.0);
    END_IF;
  END_FOR;
  bus1Applied := TRUE;
  SetpointApplied := TRUE;
ELSE
  GVL.UseTempBus1Direct := FALSE;
END_IF;

(* ---- Falling edge: clear temp inputs and deactivate ---- *)
IF NOT Enable AND Enable_Prev THEN
  GVL.UseTempGroupInputs := FALSE;
  GVL.UseTempBus1Direct := FALSE;
  MEMSET(ADR(GVL.TempGroupInput), 0, SIZEOF(GVL.TempGroupInput));
  MEMSET(ADR(GVL.TempBus1VoutSetpoint), 0, SIZEOF(GVL.TempBus1VoutSetpoint));
  MEMSET(ADR(GVL.TempBus1IoutSetpoint), 0, SIZEOF(GVL.TempBus1IoutSetpoint));
  MEMSET(ADR(GVL.TempBus1Flags), 0, SIZEOF(GVL.TempBus1Flags));
  MEMSET(ADR(GVL.TempBus1VoutSetMin), 0, SIZEOF(GVL.TempBus1VoutSetMin));
  MEMSET(ADR(GVL.TempBus1VoutSetMax), 0, SIZEOF(GVL.TempBus1VoutSetMax));
  MEMSET(ADR(GVL.TempBus1IoutSetMin), 0, SIZEOF(GVL.TempBus1IoutSetMin));
  MEMSET(ADR(GVL.TempBus1IoutSetMax), 0, SIZEOF(GVL.TempBus1IoutSetMax));
  IF bus1Applied THEN
    FOR busDev := 0 TO 3 DO
      IF (Bus1DeviceMask AND SHL(16#01, busDev)) <> 0 THEN
        GVL.OutputOn[busDev] := FALSE;
        GVL.OperationOn[busDev] := FALSE;
        GVL.Voltage[busDev] := FALSE;
        GVL.Current[busDev] := FALSE;
      END_IF;
    END_FOR;
    bus1Applied := FALSE;
  END_IF;
  SetpointApplied := FALSE;
END_IF;

Enable_Prev := Enable;

END_PROGRAM
